SYSTEM FillingCellFixed (* FillingCell (production, OPC UA driven), FillingCellDemo (self-running), SkillBench and PatternDemo run on one FORTE_PC device; PiIoConfig is for a Raspberry Pi *)
  (* Standard: 61499-2 *)
  APPLICATION FillingCell (* Production cell driven over OPC UA (/Objects/FillingCell/Filler). IoBackend 0 = simulated (force Observer.Sim_* ), 1 = GPIO (add PiIoConfig), 2 = Modbus (4diac/tools/cell_sim.py) *)
    FBS
      Boot : iec61499::events::E_RESTART;
      Observer : fillingcell::UNIT_Observer(UaRoot := "/Objects/FillingCell/Filler", UaEnable := TRUE, IoBackend := 0, NeedleUp_Gpio := 'FC_NeedleUp', NeedleUp_Modbus := "modbus[127.0.0.1:1502:1:50:d0:]", NeedleDown_Gpio := 'FC_NeedleDown', NeedleDown_Modbus := "modbus[127.0.0.1:1502:1:50:d1:]", VialPresent_Gpio := 'FC_VialPresent', VialPresent_Modbus := "modbus[127.0.0.1:1502:1:50:d2:]", Stoppered_Gpio := 'FC_Stoppered', Stoppered_Modbus := "modbus[127.0.0.1:1502:1:50:d3:]", Checked_Gpio := 'FC_Checked', Checked_Modbus := "modbus[127.0.0.1:1502:1:50:d4:]", DoorClosed_Gpio := 'FC_DoorClosed', DoorClosed_Modbus := "modbus[127.0.0.1:1502:1:50:d5:]", FilledMl_Gpio := '', FilledMl_Modbus := "modbus[127.0.0.1:1502:1:50:i0:]", Sim_NeedleUp := TRUE, Sim_VialPresent := TRUE, Sim_DoorClosed := TRUE);
      UaFacade : fillingcell::UNIT_Facade(UaRoot := "/Objects/FillingCell/Filler", UaEnable := TRUE);
      Occupation : fillingcell::FC_Occupation;
      Unit : fillingcell::FC_Unit;
      Facade : fillingcell::FC_ProcedureFacade;
    END_FBS
    SUBAPPLICATION EM_Filler (* Equipment module: one composite per skill, chained for status; instances and chain may be changed online while the unit is quiescent *)
      EVENT_INPUT
        INIT;
        UNIT_CTL WITH ControlCode;
        UNIT_STAT WITH UnitRunning, UnitQuiescent, UnitState, Mode, Owner, RemoteAllowed;
        SAMPLE WITH Cell;
        CALL_MoveDown WITH P1_MoveDown, P2_MoveDown, P3_MoveDown, P4_MoveDown;
        CALL_Dose WITH P1_Dose, P2_Dose, P3_Dose, P4_Dose;
        CALL_MoveUp WITH P1_MoveUp, P2_MoveUp, P3_MoveUp, P4_MoveUp;
        CALL_Stopper WITH P1_Stopper, P2_Stopper, P3_Stopper, P4_Stopper;
        CALL_Inspect WITH P1_Inspect, P2_Inspect, P3_Inspect, P4_Inspect;
      END_EVENT
      EVENT_OUTPUT
        INITO;
        STAT_OUT WITH Busy, HeldAll, RunAll;
        DONE_MoveDown;
        DONE_Dose;
        DONE_MoveUp;
        DONE_Stopper;
        DONE_Inspect;
        FAILED_MoveDown WITH CallError_MoveDown;
        FAILED_Dose WITH CallError_Dose;
        FAILED_MoveUp WITH CallError_MoveUp;
        FAILED_Stopper WITH CallError_Stopper;
        FAILED_Inspect WITH CallError_Inspect;
      END_EVENT
      VAR_INPUT
        ControlCode : USINT;
        UnitRunning : BOOL;
        UnitQuiescent : BOOL;
        UnitState : USINT;
        Mode : USINT;
        Owner : UDINT;
        RemoteAllowed : BOOL;
        Cell : fillingcell::ST_CellState;
        P1_MoveDown : LREAL;
        P2_MoveDown : LREAL;
        P3_MoveDown : LREAL;
        P4_MoveDown : LREAL;
        P1_Dose : LREAL;
        P2_Dose : LREAL;
        P3_Dose : LREAL;
        P4_Dose : LREAL;
        P1_MoveUp : LREAL;
        P2_MoveUp : LREAL;
        P3_MoveUp : LREAL;
        P4_MoveUp : LREAL;
        P1_Stopper : LREAL;
        P2_Stopper : LREAL;
        P3_Stopper : LREAL;
        P4_Stopper : LREAL;
        P1_Inspect : LREAL;
        P2_Inspect : LREAL;
        P3_Inspect : LREAL;
        P4_Inspect : LREAL;
      END_VAR
      VAR_OUTPUT
        Busy : BOOL;
        HeldAll : BOOL;
        RunAll : BOOL;
        CallError_MoveDown : UINT;
        CallError_Dose : UINT;
        CallError_MoveUp : UINT;
        CallError_Stopper : UINT;
        CallError_Inspect : UINT;
        Drive_MoveDown : BOOL;
        Drive_Dose : BOOL;
        Drive_MoveUp : BOOL;
        Drive_Stopper : BOOL;
        Drive_Inspect : BOOL;
      END_VAR
      FBS
        MoveDown : fillingcell::SK_MoveDown(UaRoot := "/Objects/FillingCell/Filler/Skills/MoveDown", UaEnable := TRUE, IoBackend := 0, DoGpio := 'FC_MoveDown', DoModbus := "modbus[127.0.0.1:1502:1:0::c0]");
        Dose : fillingcell::SK_Dose(UaRoot := "/Objects/FillingCell/Filler/Skills/Dose", UaEnable := TRUE, IoBackend := 0, DoGpio := 'FC_Dose', DoModbus := "modbus[127.0.0.1:1502:1:0::c1]");
        MoveUp : fillingcell::SK_MoveUp(UaRoot := "/Objects/FillingCell/Filler/Skills/MoveUp", UaEnable := TRUE, IoBackend := 0, DoGpio := 'FC_MoveUp', DoModbus := "modbus[127.0.0.1:1502:1:0::c2]");
        Stopper : fillingcell::SK_Stopper(UaRoot := "/Objects/FillingCell/Filler/Skills/Stopper", UaEnable := TRUE, IoBackend := 0, DoGpio := 'FC_Stopper', DoModbus := "modbus[127.0.0.1:1502:1:0::c3]");
        Inspect : fillingcell::SK_Inspect(UaRoot := "/Objects/FillingCell/Filler/Skills/Inspect", UaEnable := TRUE, IoBackend := 0, DoGpio := 'FC_Inspect', DoModbus := "modbus[127.0.0.1:1502:1:0::c4]");
      END_FBS
      EVENT_CONNECTIONS
        INIT TO MoveDown.INIT;
        MoveDown.INITO TO Dose.INIT;
        MoveDown.STAT_OUT TO Dose.STAT_IN;
        Dose.INITO TO MoveUp.INIT;
        Dose.STAT_OUT TO MoveUp.STAT_IN;
        MoveUp.INITO TO Stopper.INIT;
        MoveUp.STAT_OUT TO Stopper.STAT_IN;
        Stopper.INITO TO Inspect.INIT;
        Stopper.STAT_OUT TO Inspect.STAT_IN;
        Inspect.INITO TO INITO;
        Inspect.STAT_OUT TO STAT_OUT;
        UNIT_CTL TO MoveDown.UNIT_CTL;
        UNIT_STAT TO MoveDown.UNIT_STAT;
        SAMPLE TO MoveDown.SAMPLE;
        CALL_MoveDown TO MoveDown.CALL;
        MoveDown.DONE TO DONE_MoveDown;
        MoveDown.FAILED TO FAILED_MoveDown;
        UNIT_CTL TO Dose.UNIT_CTL;
        UNIT_STAT TO Dose.UNIT_STAT;
        SAMPLE TO Dose.SAMPLE;
        CALL_Dose TO Dose.CALL;
        Dose.DONE TO DONE_Dose;
        Dose.FAILED TO FAILED_Dose;
        UNIT_CTL TO MoveUp.UNIT_CTL;
        UNIT_STAT TO MoveUp.UNIT_STAT;
        SAMPLE TO MoveUp.SAMPLE;
        CALL_MoveUp TO MoveUp.CALL;
        MoveUp.DONE TO DONE_MoveUp;
        MoveUp.FAILED TO FAILED_MoveUp;
        UNIT_CTL TO Stopper.UNIT_CTL;
        UNIT_STAT TO Stopper.UNIT_STAT;
        SAMPLE TO Stopper.SAMPLE;
        CALL_Stopper TO Stopper.CALL;
        Stopper.DONE TO DONE_Stopper;
        Stopper.FAILED TO FAILED_Stopper;
        UNIT_CTL TO Inspect.UNIT_CTL;
        UNIT_STAT TO Inspect.UNIT_STAT;
        SAMPLE TO Inspect.SAMPLE;
        CALL_Inspect TO Inspect.CALL;
        Inspect.DONE TO DONE_Inspect;
        Inspect.FAILED TO FAILED_Inspect;
      END_CONNECTIONS
      DATA_CONNECTIONS
        MoveDown.BusyOut TO Dose.BusyIn;
        MoveDown.HeldOut TO Dose.HeldIn;
        MoveDown.RunOut TO Dose.RunIn;
        Dose.BusyOut TO MoveUp.BusyIn;
        Dose.HeldOut TO MoveUp.HeldIn;
        Dose.RunOut TO MoveUp.RunIn;
        MoveUp.BusyOut TO Stopper.BusyIn;
        MoveUp.HeldOut TO Stopper.HeldIn;
        MoveUp.RunOut TO Stopper.RunIn;
        Stopper.BusyOut TO Inspect.BusyIn;
        Stopper.HeldOut TO Inspect.HeldIn;
        Stopper.RunOut TO Inspect.RunIn;
        Inspect.BusyOut TO Busy;
        Inspect.HeldOut TO HeldAll;
        Inspect.RunOut TO RunAll;
        ControlCode TO MoveDown.ControlCode;
        Cell TO MoveDown.Cell;
        MoveDown.CallError TO CallError_MoveDown;
        MoveDown.Drive TO Drive_MoveDown;
        UnitRunning TO MoveDown.UnitRunning;
        UnitQuiescent TO MoveDown.UnitQuiescent;
        UnitState TO MoveDown.UnitState;
        Mode TO MoveDown.Mode;
        Owner TO MoveDown.Owner;
        RemoteAllowed TO MoveDown.RemoteAllowed;
        P1_MoveDown TO MoveDown.P1;
        P2_MoveDown TO MoveDown.P2;
        P3_MoveDown TO MoveDown.P3;
        P4_MoveDown TO MoveDown.P4;
        ControlCode TO Dose.ControlCode;
        Cell TO Dose.Cell;
        Dose.CallError TO CallError_Dose;
        Dose.Drive TO Drive_Dose;
        UnitRunning TO Dose.UnitRunning;
        UnitQuiescent TO Dose.UnitQuiescent;
        UnitState TO Dose.UnitState;
        Mode TO Dose.Mode;
        Owner TO Dose.Owner;
        RemoteAllowed TO Dose.RemoteAllowed;
        P1_Dose TO Dose.P1;
        P2_Dose TO Dose.P2;
        P3_Dose TO Dose.P3;
        P4_Dose TO Dose.P4;
        ControlCode TO MoveUp.ControlCode;
        Cell TO MoveUp.Cell;
        MoveUp.CallError TO CallError_MoveUp;
        MoveUp.Drive TO Drive_MoveUp;
        UnitRunning TO MoveUp.UnitRunning;
        UnitQuiescent TO MoveUp.UnitQuiescent;
        UnitState TO MoveUp.UnitState;
        Mode TO MoveUp.Mode;
        Owner TO MoveUp.Owner;
        RemoteAllowed TO MoveUp.RemoteAllowed;
        P1_MoveUp TO MoveUp.P1;
        P2_MoveUp TO MoveUp.P2;
        P3_MoveUp TO MoveUp.P3;
        P4_MoveUp TO MoveUp.P4;
        ControlCode TO Stopper.ControlCode;
        Cell TO Stopper.Cell;
        Stopper.CallError TO CallError_Stopper;
        Stopper.Drive TO Drive_Stopper;
        UnitRunning TO Stopper.UnitRunning;
        UnitQuiescent TO Stopper.UnitQuiescent;
        UnitState TO Stopper.UnitState;
        Mode TO Stopper.Mode;
        Owner TO Stopper.Owner;
        RemoteAllowed TO Stopper.RemoteAllowed;
        P1_Stopper TO Stopper.P1;
        P2_Stopper TO Stopper.P2;
        P3_Stopper TO Stopper.P3;
        P4_Stopper TO Stopper.P4;
        ControlCode TO Inspect.ControlCode;
        Cell TO Inspect.Cell;
        Inspect.CallError TO CallError_Inspect;
        Inspect.Drive TO Drive_Inspect;
        UnitRunning TO Inspect.UnitRunning;
        UnitQuiescent TO Inspect.UnitQuiescent;
        UnitState TO Inspect.UnitState;
        Mode TO Inspect.Mode;
        Owner TO Inspect.Owner;
        RemoteAllowed TO Inspect.RemoteAllowed;
        P1_Inspect TO Inspect.P1;
        P2_Inspect TO Inspect.P2;
        P3_Inspect TO Inspect.P3;
        P4_Inspect TO Inspect.P4;
      END_CONNECTIONS
    END_SUBAPPLICATION
    SUBAPPLICATION PROC (* INTENTIONALLY EMPTY: generated procedure (P_* pattern instances) calls skills via CALL_*/DONE_*/FAILED_* *)
      EVENT_INPUT
        START;
        RESET;
        CMD WITH Command;
        DONE_MoveDown;
        DONE_Dose;
        DONE_MoveUp;
        DONE_Stopper;
        DONE_Inspect;
        FAILED_MoveDown WITH CallError_MoveDown;
        FAILED_Dose WITH CallError_Dose;
        FAILED_MoveUp WITH CallError_MoveUp;
        FAILED_Stopper WITH CallError_Stopper;
        FAILED_Inspect WITH CallError_Inspect;
      END_EVENT
      EVENT_OUTPUT
        FINISHED;
        FAILED;
        CALL_MoveDown WITH P1_MoveDown, P2_MoveDown, P3_MoveDown, P4_MoveDown;
        CALL_Dose WITH P1_Dose, P2_Dose, P3_Dose, P4_Dose;
        CALL_MoveUp WITH P1_MoveUp, P2_MoveUp, P3_MoveUp, P4_MoveUp;
        CALL_Stopper WITH P1_Stopper, P2_Stopper, P3_Stopper, P4_Stopper;
        CALL_Inspect WITH P1_Inspect, P2_Inspect, P3_Inspect, P4_Inspect;
      END_EVENT
      VAR_INPUT
        Command : USINT;
        CallError_MoveDown : UINT;
        CallError_Dose : UINT;
        CallError_MoveUp : UINT;
        CallError_Stopper : UINT;
        CallError_Inspect : UINT;
      END_VAR
      VAR_OUTPUT
        P1_MoveDown : LREAL;
        P2_MoveDown : LREAL;
        P3_MoveDown : LREAL;
        P4_MoveDown : LREAL;
        P1_Dose : LREAL;
        P2_Dose : LREAL;
        P3_Dose : LREAL;
        P4_Dose : LREAL;
        P1_MoveUp : LREAL;
        P2_MoveUp : LREAL;
        P3_MoveUp : LREAL;
        P4_MoveUp : LREAL;
        P1_Stopper : LREAL;
        P2_Stopper : LREAL;
        P3_Stopper : LREAL;
        P4_Stopper : LREAL;
        P1_Inspect : LREAL;
        P2_Inspect : LREAL;
        P3_Inspect : LREAL;
        P4_Inspect : LREAL;
      END_VAR
    END_SUBAPPLICATION
    EVENT_CONNECTIONS
      Boot.COLD TO Observer.INIT;
      Boot.WARM TO Observer.INIT;
      Unit.CNF TO EM_Filler.UNIT_STAT;
      Occupation.CNF TO EM_Filler.UNIT_STAT;
      Unit.CONTROL TO EM_Filler.UNIT_CTL;
      EM_Filler.STAT_OUT TO Unit.STATUS;
      Observer.SAMPLE TO EM_Filler.SAMPLE;
      Observer.UNSAFE TO Unit.UNSAFE;
      Unit.PROC_CMD TO Facade.CMD;
      Facade.EXEC TO PROC.CMD;
      Facade.START TO PROC.START;
      Facade.RESET TO PROC.RESET;
      PROC.FINISHED TO Facade.FINISHED;
      PROC.FAILED TO Facade.FAILED;
      Facade.DONE TO Unit.PROC_DONE;
      Facade.FAULT TO Unit.FAULT;
      PROC.CALL_MoveDown TO EM_Filler.CALL_MoveDown;
      EM_Filler.DONE_MoveDown TO PROC.DONE_MoveDown;
      EM_Filler.FAILED_MoveDown TO PROC.FAILED_MoveDown;
      PROC.CALL_Dose TO EM_Filler.CALL_Dose;
      EM_Filler.DONE_Dose TO PROC.DONE_Dose;
      EM_Filler.FAILED_Dose TO PROC.FAILED_Dose;
      PROC.CALL_MoveUp TO EM_Filler.CALL_MoveUp;
      EM_Filler.DONE_MoveUp TO PROC.DONE_MoveUp;
      EM_Filler.FAILED_MoveUp TO PROC.FAILED_MoveUp;
      PROC.CALL_Stopper TO EM_Filler.CALL_Stopper;
      EM_Filler.DONE_Stopper TO PROC.DONE_Stopper;
      EM_Filler.FAILED_Stopper TO PROC.FAILED_Stopper;
      PROC.CALL_Inspect TO EM_Filler.CALL_Inspect;
      EM_Filler.DONE_Inspect TO PROC.DONE_Inspect;
      EM_Filler.FAILED_Inspect TO PROC.FAILED_Inspect;
      Observer.INITO TO UaFacade.INIT;
      UaFacade.INITO TO EM_Filler.INIT;
      UaFacade.U_CMD TO Unit.CMD;
      UaFacade.O_CMD TO Occupation.CMD;
      Unit.CMD_ACK TO UaFacade.U_ACK;
      Unit.CMD_REJ TO UaFacade.U_REJ;
      Occupation.CNF TO UaFacade.O_ACK;
      Occupation.REJECTED TO UaFacade.O_REJ;
      Unit.CNF TO UaFacade.PUB;
      Occupation.CNF TO UaFacade.PUB;
    END_CONNECTIONS
    DATA_CONNECTIONS
      Occupation.Owner TO Unit.Owner;
      Occupation.RemoteAllowed TO Unit.RemoteAllowed;
      Occupation.Owner TO EM_Filler.Owner;
      Occupation.RemoteAllowed TO EM_Filler.RemoteAllowed;
      Unit.Running TO EM_Filler.UnitRunning;
      Unit.Quiescent TO EM_Filler.UnitQuiescent;
      Unit.State TO EM_Filler.UnitState;
      Unit.Mode TO EM_Filler.Mode;
      Unit.ControlCode TO EM_Filler.ControlCode;
      Unit.Quiescent TO Occupation.Quiescent;
      Unit.Quiescent TO Facade.Quiescent;
      EM_Filler.Busy TO Unit.Busy;
      EM_Filler.HeldAll TO Unit.HeldAll;
      EM_Filler.RunAll TO Unit.RunAll;
      Observer.Cell TO EM_Filler.Cell;
      Observer.Safe TO Unit.Safe;
      Unit.ProcedureCommand TO Facade.Command;
      Facade.CommandOut TO PROC.Command;
      Facade.Ready TO Unit.ProcedureReady;
      PROC.P1_MoveDown TO EM_Filler.P1_MoveDown;
      PROC.P2_MoveDown TO EM_Filler.P2_MoveDown;
      PROC.P3_MoveDown TO EM_Filler.P3_MoveDown;
      PROC.P4_MoveDown TO EM_Filler.P4_MoveDown;
      EM_Filler.CallError_MoveDown TO PROC.CallError_MoveDown;
      PROC.P1_Dose TO EM_Filler.P1_Dose;
      PROC.P2_Dose TO EM_Filler.P2_Dose;
      PROC.P3_Dose TO EM_Filler.P3_Dose;
      PROC.P4_Dose TO EM_Filler.P4_Dose;
      EM_Filler.CallError_Dose TO PROC.CallError_Dose;
      PROC.P1_MoveUp TO EM_Filler.P1_MoveUp;
      PROC.P2_MoveUp TO EM_Filler.P2_MoveUp;
      PROC.P3_MoveUp TO EM_Filler.P3_MoveUp;
      PROC.P4_MoveUp TO EM_Filler.P4_MoveUp;
      EM_Filler.CallError_MoveUp TO PROC.CallError_MoveUp;
      PROC.P1_Stopper TO EM_Filler.P1_Stopper;
      PROC.P2_Stopper TO EM_Filler.P2_Stopper;
      PROC.P3_Stopper TO EM_Filler.P3_Stopper;
      PROC.P4_Stopper TO EM_Filler.P4_Stopper;
      EM_Filler.CallError_Stopper TO PROC.CallError_Stopper;
      PROC.P1_Inspect TO EM_Filler.P1_Inspect;
      PROC.P2_Inspect TO EM_Filler.P2_Inspect;
      PROC.P3_Inspect TO EM_Filler.P3_Inspect;
      PROC.P4_Inspect TO EM_Filler.P4_Inspect;
      EM_Filler.CallError_Inspect TO PROC.CallError_Inspect;
      UaFacade.Requester TO Unit.Requester;
      UaFacade.Requester TO Occupation.Requester;
      UaFacade.U_Code TO Unit.Command;
      UaFacade.U_Mode TO Unit.RequestedMode;
      UaFacade.O_Code TO Occupation.Command;
      Unit.State TO UaFacade.UnitState;
      Unit.Mode TO UaFacade.UnitMode;
      Occupation.State TO UaFacade.OccState;
      Occupation.Owner TO UaFacade.Owner;
    END_CONNECTIONS
  END_APPLICATION
  APPLICATION FillingCellDemo (* Self-running demo: plant model and automatic operator cycle the whole cell through the PROC procedure; watch Operator.Cycles, Unit.State, Plant.* in the IDE monitoring (no OPC UA: FORTE 3.3 serves OPC UA for one resource only, used by FillingCell) *)
    FBS
      Boot : iec61499::events::E_RESTART;
      Observer : fillingcell::UNIT_Observer(UaRoot := "/Objects/Demo/Filler", UaEnable := FALSE, IoBackend := 0, CycleTime := T#50ms);
      Occupation : fillingcell::FC_Occupation;
      Unit : fillingcell::FC_Unit;
      Facade : fillingcell::FC_ProcedureFacade(Installed := TRUE);
      Plant : fillingcell::DEMO_Plant;
      PlantClock : iec61499::events::E_CYCLE(DT := T#20ms);
      Operator : fillingcell::DEMO_Operator;
      OpDelay : iec61499::events::E_DELAY;
    END_FBS
    SUBAPPLICATION EM_Filler (* Equipment module: one composite per skill, chained for status; instances and chain may be changed online while the unit is quiescent *)
      EVENT_INPUT
        INIT;
        UNIT_CTL WITH ControlCode;
        UNIT_STAT WITH UnitRunning, UnitQuiescent, UnitState, Mode, Owner, RemoteAllowed;
        SAMPLE WITH Cell;
        CALL_MoveDown WITH P1_MoveDown, P2_MoveDown, P3_MoveDown, P4_MoveDown;
        CALL_Dose WITH P1_Dose, P2_Dose, P3_Dose, P4_Dose;
        CALL_MoveUp WITH P1_MoveUp, P2_MoveUp, P3_MoveUp, P4_MoveUp;
        CALL_Stopper WITH P1_Stopper, P2_Stopper, P3_Stopper, P4_Stopper;
        CALL_Inspect WITH P1_Inspect, P2_Inspect, P3_Inspect, P4_Inspect;
      END_EVENT
      EVENT_OUTPUT
        INITO;
        STAT_OUT WITH Busy, HeldAll, RunAll;
        DONE_MoveDown;
        DONE_Dose;
        DONE_MoveUp;
        DONE_Stopper;
        DONE_Inspect;
        FAILED_MoveDown WITH CallError_MoveDown;
        FAILED_Dose WITH CallError_Dose;
        FAILED_MoveUp WITH CallError_MoveUp;
        FAILED_Stopper WITH CallError_Stopper;
        FAILED_Inspect WITH CallError_Inspect;
      END_EVENT
      VAR_INPUT
        ControlCode : USINT;
        UnitRunning : BOOL;
        UnitQuiescent : BOOL;
        UnitState : USINT;
        Mode : USINT;
        Owner : UDINT;
        RemoteAllowed : BOOL;
        Cell : fillingcell::ST_CellState;
        P1_MoveDown : LREAL;
        P2_MoveDown : LREAL;
        P3_MoveDown : LREAL;
        P4_MoveDown : LREAL;
        P1_Dose : LREAL;
        P2_Dose : LREAL;
        P3_Dose : LREAL;
        P4_Dose : LREAL;
        P1_MoveUp : LREAL;
        P2_MoveUp : LREAL;
        P3_MoveUp : LREAL;
        P4_MoveUp : LREAL;
        P1_Stopper : LREAL;
        P2_Stopper : LREAL;
        P3_Stopper : LREAL;
        P4_Stopper : LREAL;
        P1_Inspect : LREAL;
        P2_Inspect : LREAL;
        P3_Inspect : LREAL;
        P4_Inspect : LREAL;
      END_VAR
      VAR_OUTPUT
        Busy : BOOL;
        HeldAll : BOOL;
        RunAll : BOOL;
        CallError_MoveDown : UINT;
        CallError_Dose : UINT;
        CallError_MoveUp : UINT;
        CallError_Stopper : UINT;
        CallError_Inspect : UINT;
        Drive_MoveDown : BOOL;
        Drive_Dose : BOOL;
        Drive_MoveUp : BOOL;
        Drive_Stopper : BOOL;
        Drive_Inspect : BOOL;
      END_VAR
      FBS
        MoveDown : fillingcell::SK_MoveDown(UaRoot := "/Objects/Demo/Filler/Skills/MoveDown", UaEnable := FALSE, IoBackend := 0);
        Dose : fillingcell::SK_Dose(UaRoot := "/Objects/Demo/Filler/Skills/Dose", UaEnable := FALSE, IoBackend := 0);
        MoveUp : fillingcell::SK_MoveUp(UaRoot := "/Objects/Demo/Filler/Skills/MoveUp", UaEnable := FALSE, IoBackend := 0);
        Stopper : fillingcell::SK_Stopper(UaRoot := "/Objects/Demo/Filler/Skills/Stopper", UaEnable := FALSE, IoBackend := 0);
        Inspect : fillingcell::SK_Inspect(UaRoot := "/Objects/Demo/Filler/Skills/Inspect", UaEnable := FALSE, IoBackend := 0);
      END_FBS
      EVENT_CONNECTIONS
        INIT TO MoveDown.INIT;
        MoveDown.INITO TO Dose.INIT;
        MoveDown.STAT_OUT TO Dose.STAT_IN;
        Dose.INITO TO MoveUp.INIT;
        Dose.STAT_OUT TO MoveUp.STAT_IN;
        MoveUp.INITO TO Stopper.INIT;
        MoveUp.STAT_OUT TO Stopper.STAT_IN;
        Stopper.INITO TO Inspect.INIT;
        Stopper.STAT_OUT TO Inspect.STAT_IN;
        Inspect.INITO TO INITO;
        Inspect.STAT_OUT TO STAT_OUT;
        UNIT_CTL TO MoveDown.UNIT_CTL;
        UNIT_STAT TO MoveDown.UNIT_STAT;
        SAMPLE TO MoveDown.SAMPLE;
        CALL_MoveDown TO MoveDown.CALL;
        MoveDown.DONE TO DONE_MoveDown;
        MoveDown.FAILED TO FAILED_MoveDown;
        UNIT_CTL TO Dose.UNIT_CTL;
        UNIT_STAT TO Dose.UNIT_STAT;
        SAMPLE TO Dose.SAMPLE;
        CALL_Dose TO Dose.CALL;
        Dose.DONE TO DONE_Dose;
        Dose.FAILED TO FAILED_Dose;
        UNIT_CTL TO MoveUp.UNIT_CTL;
        UNIT_STAT TO MoveUp.UNIT_STAT;
        SAMPLE TO MoveUp.SAMPLE;
        CALL_MoveUp TO MoveUp.CALL;
        MoveUp.DONE TO DONE_MoveUp;
        MoveUp.FAILED TO FAILED_MoveUp;
        UNIT_CTL TO Stopper.UNIT_CTL;
        UNIT_STAT TO Stopper.UNIT_STAT;
        SAMPLE TO Stopper.SAMPLE;
        CALL_Stopper TO Stopper.CALL;
        Stopper.DONE TO DONE_Stopper;
        Stopper.FAILED TO FAILED_Stopper;
        UNIT_CTL TO Inspect.UNIT_CTL;
        UNIT_STAT TO Inspect.UNIT_STAT;
        SAMPLE TO Inspect.SAMPLE;
        CALL_Inspect TO Inspect.CALL;
        Inspect.DONE TO DONE_Inspect;
        Inspect.FAILED TO FAILED_Inspect;
      END_CONNECTIONS
      DATA_CONNECTIONS
        MoveDown.BusyOut TO Dose.BusyIn;
        MoveDown.HeldOut TO Dose.HeldIn;
        MoveDown.RunOut TO Dose.RunIn;
        Dose.BusyOut TO MoveUp.BusyIn;
        Dose.HeldOut TO MoveUp.HeldIn;
        Dose.RunOut TO MoveUp.RunIn;
        MoveUp.BusyOut TO Stopper.BusyIn;
        MoveUp.HeldOut TO Stopper.HeldIn;
        MoveUp.RunOut TO Stopper.RunIn;
        Stopper.BusyOut TO Inspect.BusyIn;
        Stopper.HeldOut TO Inspect.HeldIn;
        Stopper.RunOut TO Inspect.RunIn;
        Inspect.BusyOut TO Busy;
        Inspect.HeldOut TO HeldAll;
        Inspect.RunOut TO RunAll;
        ControlCode TO MoveDown.ControlCode;
        Cell TO MoveDown.Cell;
        MoveDown.CallError TO CallError_MoveDown;
        MoveDown.Drive TO Drive_MoveDown;
        UnitRunning TO MoveDown.UnitRunning;
        UnitQuiescent TO MoveDown.UnitQuiescent;
        UnitState TO MoveDown.UnitState;
        Mode TO MoveDown.Mode;
        Owner TO MoveDown.Owner;
        RemoteAllowed TO MoveDown.RemoteAllowed;
        P1_MoveDown TO MoveDown.P1;
        P2_MoveDown TO MoveDown.P2;
        P3_MoveDown TO MoveDown.P3;
        P4_MoveDown TO MoveDown.P4;
        ControlCode TO Dose.ControlCode;
        Cell TO Dose.Cell;
        Dose.CallError TO CallError_Dose;
        Dose.Drive TO Drive_Dose;
        UnitRunning TO Dose.UnitRunning;
        UnitQuiescent TO Dose.UnitQuiescent;
        UnitState TO Dose.UnitState;
        Mode TO Dose.Mode;
        Owner TO Dose.Owner;
        RemoteAllowed TO Dose.RemoteAllowed;
        P1_Dose TO Dose.P1;
        P2_Dose TO Dose.P2;
        P3_Dose TO Dose.P3;
        P4_Dose TO Dose.P4;
        ControlCode TO MoveUp.ControlCode;
        Cell TO MoveUp.Cell;
        MoveUp.CallError TO CallError_MoveUp;
        MoveUp.Drive TO Drive_MoveUp;
        UnitRunning TO MoveUp.UnitRunning;
        UnitQuiescent TO MoveUp.UnitQuiescent;
        UnitState TO MoveUp.UnitState;
        Mode TO MoveUp.Mode;
        Owner TO MoveUp.Owner;
        RemoteAllowed TO MoveUp.RemoteAllowed;
        P1_MoveUp TO MoveUp.P1;
        P2_MoveUp TO MoveUp.P2;
        P3_MoveUp TO MoveUp.P3;
        P4_MoveUp TO MoveUp.P4;
        ControlCode TO Stopper.ControlCode;
        Cell TO Stopper.Cell;
        Stopper.CallError TO CallError_Stopper;
        Stopper.Drive TO Drive_Stopper;
        UnitRunning TO Stopper.UnitRunning;
        UnitQuiescent TO Stopper.UnitQuiescent;
        UnitState TO Stopper.UnitState;
        Mode TO Stopper.Mode;
        Owner TO Stopper.Owner;
        RemoteAllowed TO Stopper.RemoteAllowed;
        P1_Stopper TO Stopper.P1;
        P2_Stopper TO Stopper.P2;
        P3_Stopper TO Stopper.P3;
        P4_Stopper TO Stopper.P4;
        ControlCode TO Inspect.ControlCode;
        Cell TO Inspect.Cell;
        Inspect.CallError TO CallError_Inspect;
        Inspect.Drive TO Drive_Inspect;
        UnitRunning TO Inspect.UnitRunning;
        UnitQuiescent TO Inspect.UnitQuiescent;
        UnitState TO Inspect.UnitState;
        Mode TO Inspect.Mode;
        Owner TO Inspect.Owner;
        RemoteAllowed TO Inspect.RemoteAllowed;
        P1_Inspect TO Inspect.P1;
        P2_Inspect TO Inspect.P2;
        P3_Inspect TO Inspect.P3;
        P4_Inspect TO Inspect.P4;
      END_CONNECTIONS
    END_SUBAPPLICATION
    SUBAPPLICATION PROC (* Demo procedure: MoveDown, Dose x2 (P_Loop), MoveUp, Stopper, Inspect *)
      EVENT_INPUT
        START;
        RESET;
        CMD WITH Command;
        DONE_MoveDown;
        DONE_Dose;
        DONE_MoveUp;
        DONE_Stopper;
        DONE_Inspect;
        FAILED_MoveDown WITH CallError_MoveDown;
        FAILED_Dose WITH CallError_Dose;
        FAILED_MoveUp WITH CallError_MoveUp;
        FAILED_Stopper WITH CallError_Stopper;
        FAILED_Inspect WITH CallError_Inspect;
      END_EVENT
      EVENT_OUTPUT
        FINISHED;
        FAILED;
        CALL_MoveDown WITH P1_MoveDown, P2_MoveDown, P3_MoveDown, P4_MoveDown;
        CALL_Dose WITH P1_Dose, P2_Dose, P3_Dose, P4_Dose;
        CALL_MoveUp WITH P1_MoveUp, P2_MoveUp, P3_MoveUp, P4_MoveUp;
        CALL_Stopper WITH P1_Stopper, P2_Stopper, P3_Stopper, P4_Stopper;
        CALL_Inspect WITH P1_Inspect, P2_Inspect, P3_Inspect, P4_Inspect;
      END_EVENT
      VAR_INPUT
        Command : USINT;
        CallError_MoveDown : UINT;
        CallError_Dose : UINT;
        CallError_MoveUp : UINT;
        CallError_Stopper : UINT;
        CallError_Inspect : UINT;
      END_VAR
      VAR_OUTPUT
        P1_MoveDown : LREAL;
        P2_MoveDown : LREAL;
        P3_MoveDown : LREAL;
        P4_MoveDown : LREAL;
        P1_Dose : LREAL;
        P2_Dose : LREAL;
        P3_Dose : LREAL;
        P4_Dose : LREAL;
        P1_MoveUp : LREAL;
        P2_MoveUp : LREAL;
        P3_MoveUp : LREAL;
        P4_MoveUp : LREAL;
        P1_Stopper : LREAL;
        P2_Stopper : LREAL;
        P3_Stopper : LREAL;
        P4_Stopper : LREAL;
        P1_Inspect : LREAL;
        P2_Inspect : LREAL;
        P3_Inspect : LREAL;
        P4_Inspect : LREAL;
      END_VAR
      FBS
        MoveDown : fillingcell::P_Call;
        Dose : fillingcell::P_Call(P1 := 0.3);
        MoveUp : fillingcell::P_Call;
        Stopper : fillingcell::P_Call;
        Inspect : fillingcell::P_Call;
        DoseLoop : fillingcell::P_Loop(Count := 2);
      END_FBS
      EVENT_CONNECTIONS
        START TO MoveDown.EI;
        MoveDown.EO TO DoseLoop.EI;
        DoseLoop.BODY TO Dose.EI;
        Dose.EO TO DoseLoop.NEXT;
        DoseLoop.EO TO MoveUp.EI;
        MoveUp.EO TO Stopper.EI;
        Stopper.EO TO Inspect.EI;
        Inspect.EO TO FINISHED;
        RESET TO DoseLoop.RESET;
        MoveDown.CALL TO CALL_MoveDown;
        DONE_MoveDown TO MoveDown.DONE;
        FAILED_MoveDown TO MoveDown.FAILED;
        MoveDown.ERR TO FAILED;
        RESET TO MoveDown.RESET;
        Dose.CALL TO CALL_Dose;
        DONE_Dose TO Dose.DONE;
        FAILED_Dose TO Dose.FAILED;
        Dose.ERR TO FAILED;
        RESET TO Dose.RESET;
        MoveUp.CALL TO CALL_MoveUp;
        DONE_MoveUp TO MoveUp.DONE;
        FAILED_MoveUp TO MoveUp.FAILED;
        MoveUp.ERR TO FAILED;
        RESET TO MoveUp.RESET;
        Stopper.CALL TO CALL_Stopper;
        DONE_Stopper TO Stopper.DONE;
        FAILED_Stopper TO Stopper.FAILED;
        Stopper.ERR TO FAILED;
        RESET TO Stopper.RESET;
        Inspect.CALL TO CALL_Inspect;
        DONE_Inspect TO Inspect.DONE;
        FAILED_Inspect TO Inspect.FAILED;
        Inspect.ERR TO FAILED;
        RESET TO Inspect.RESET;
      END_CONNECTIONS
      DATA_CONNECTIONS
        Dose.CP1 TO P1_Dose;
        CallError_MoveDown TO MoveDown.CallError;
        CallError_Dose TO Dose.CallError;
        CallError_MoveUp TO MoveUp.CallError;
        CallError_Stopper TO Stopper.CallError;
        CallError_Inspect TO Inspect.CallError;
      END_CONNECTIONS
    END_SUBAPPLICATION
    EVENT_CONNECTIONS
      Boot.COLD TO Observer.INIT;
      Boot.WARM TO Observer.INIT;
      Unit.CNF TO EM_Filler.UNIT_STAT;
      Occupation.CNF TO EM_Filler.UNIT_STAT;
      Unit.CONTROL TO EM_Filler.UNIT_CTL;
      EM_Filler.STAT_OUT TO Unit.STATUS;
      Observer.SAMPLE TO EM_Filler.SAMPLE;
      Observer.UNSAFE TO Unit.UNSAFE;
      Unit.PROC_CMD TO Facade.CMD;
      Facade.EXEC TO PROC.CMD;
      Facade.START TO PROC.START;
      Facade.RESET TO PROC.RESET;
      PROC.FINISHED TO Facade.FINISHED;
      PROC.FAILED TO Facade.FAILED;
      Facade.DONE TO Unit.PROC_DONE;
      Facade.FAULT TO Unit.FAULT;
      PROC.CALL_MoveDown TO EM_Filler.CALL_MoveDown;
      EM_Filler.DONE_MoveDown TO PROC.DONE_MoveDown;
      EM_Filler.FAILED_MoveDown TO PROC.FAILED_MoveDown;
      PROC.CALL_Dose TO EM_Filler.CALL_Dose;
      EM_Filler.DONE_Dose TO PROC.DONE_Dose;
      EM_Filler.FAILED_Dose TO PROC.FAILED_Dose;
      PROC.CALL_MoveUp TO EM_Filler.CALL_MoveUp;
      EM_Filler.DONE_MoveUp TO PROC.DONE_MoveUp;
      EM_Filler.FAILED_MoveUp TO PROC.FAILED_MoveUp;
      PROC.CALL_Stopper TO EM_Filler.CALL_Stopper;
      EM_Filler.DONE_Stopper TO PROC.DONE_Stopper;
      EM_Filler.FAILED_Stopper TO PROC.FAILED_Stopper;
      PROC.CALL_Inspect TO EM_Filler.CALL_Inspect;
      EM_Filler.DONE_Inspect TO PROC.DONE_Inspect;
      EM_Filler.FAILED_Inspect TO PROC.FAILED_Inspect;
      Boot.COLD TO Plant.INIT;
      Boot.WARM TO Plant.INIT;
      Boot.COLD TO PlantClock.START;
      Boot.WARM TO PlantClock.START;
      PlantClock.EO TO Plant.TICK;
      Plant.CNF TO Observer.SIM;
      Observer.INITO TO EM_Filler.INIT;
      EM_Filler.INITO TO Facade.CONFIG;
      Facade.CNF TO Operator.START;
      Operator.O_CMD TO Occupation.CMD;
      Operator.U_CMD TO Unit.CMD;
      Operator.NEW_VIAL TO Plant.NEW_VIAL;
      Operator.WAIT TO OpDelay.START;
      OpDelay.EO TO Operator.TIMER;
      Unit.CNF TO Operator.UNIT;
      Unit.CMD_REJ TO Operator.REJ;
    END_CONNECTIONS
    DATA_CONNECTIONS
      Occupation.Owner TO Unit.Owner;
      Occupation.RemoteAllowed TO Unit.RemoteAllowed;
      Occupation.Owner TO EM_Filler.Owner;
      Occupation.RemoteAllowed TO EM_Filler.RemoteAllowed;
      Unit.Running TO EM_Filler.UnitRunning;
      Unit.Quiescent TO EM_Filler.UnitQuiescent;
      Unit.State TO EM_Filler.UnitState;
      Unit.Mode TO EM_Filler.Mode;
      Unit.ControlCode TO EM_Filler.ControlCode;
      Unit.Quiescent TO Occupation.Quiescent;
      Unit.Quiescent TO Facade.Quiescent;
      EM_Filler.Busy TO Unit.Busy;
      EM_Filler.HeldAll TO Unit.HeldAll;
      EM_Filler.RunAll TO Unit.RunAll;
      Observer.Cell TO EM_Filler.Cell;
      Observer.Safe TO Unit.Safe;
      Unit.ProcedureCommand TO Facade.Command;
      Facade.CommandOut TO PROC.Command;
      Facade.Ready TO Unit.ProcedureReady;
      PROC.P1_MoveDown TO EM_Filler.P1_MoveDown;
      PROC.P2_MoveDown TO EM_Filler.P2_MoveDown;
      PROC.P3_MoveDown TO EM_Filler.P3_MoveDown;
      PROC.P4_MoveDown TO EM_Filler.P4_MoveDown;
      EM_Filler.CallError_MoveDown TO PROC.CallError_MoveDown;
      PROC.P1_Dose TO EM_Filler.P1_Dose;
      PROC.P2_Dose TO EM_Filler.P2_Dose;
      PROC.P3_Dose TO EM_Filler.P3_Dose;
      PROC.P4_Dose TO EM_Filler.P4_Dose;
      EM_Filler.CallError_Dose TO PROC.CallError_Dose;
      PROC.P1_MoveUp TO EM_Filler.P1_MoveUp;
      PROC.P2_MoveUp TO EM_Filler.P2_MoveUp;
      PROC.P3_MoveUp TO EM_Filler.P3_MoveUp;
      PROC.P4_MoveUp TO EM_Filler.P4_MoveUp;
      EM_Filler.CallError_MoveUp TO PROC.CallError_MoveUp;
      PROC.P1_Stopper TO EM_Filler.P1_Stopper;
      PROC.P2_Stopper TO EM_Filler.P2_Stopper;
      PROC.P3_Stopper TO EM_Filler.P3_Stopper;
      PROC.P4_Stopper TO EM_Filler.P4_Stopper;
      EM_Filler.CallError_Stopper TO PROC.CallError_Stopper;
      PROC.P1_Inspect TO EM_Filler.P1_Inspect;
      PROC.P2_Inspect TO EM_Filler.P2_Inspect;
      PROC.P3_Inspect TO EM_Filler.P3_Inspect;
      PROC.P4_Inspect TO EM_Filler.P4_Inspect;
      EM_Filler.CallError_Inspect TO PROC.CallError_Inspect;
      Operator.Requester TO Unit.Requester;
      Operator.Requester TO Occupation.Requester;
      Operator.U_Code TO Unit.Command;
      Operator.U_Mode TO Unit.RequestedMode;
      Operator.O_Code TO Occupation.Command;
      Unit.State TO Operator.UnitState;
      Operator.Delay TO OpDelay.DT;
      Plant.NeedleUp TO Observer.Sim_NeedleUp;
      Plant.NeedleDown TO Observer.Sim_NeedleDown;
      Plant.VialPresent TO Observer.Sim_VialPresent;
      Plant.FilledMl TO Observer.Sim_FilledMl;
      Plant.Stoppered TO Observer.Sim_Stoppered;
      Plant.Checked TO Observer.Sim_Checked;
      Plant.DoorClosed TO Observer.Sim_DoorClosed;
      EM_Filler.Drive_MoveDown TO Plant.DriveMoveDown;
      EM_Filler.Drive_Dose TO Plant.DriveDose;
      EM_Filler.Drive_MoveUp TO Plant.DriveMoveUp;
      EM_Filler.Drive_Stopper TO Plant.DriveStopper;
      EM_Filler.Drive_Inspect TO Plant.DriveInspect;
    END_CONNECTIONS
  END_APPLICATION
  APPLICATION SkillBench (* Demo: SK_Dose is called periodically with P1 = 0.3 mL; watch Dose.State, Plant.FilledMl, Done.CV and Failed.CV in the IDE monitoring *)
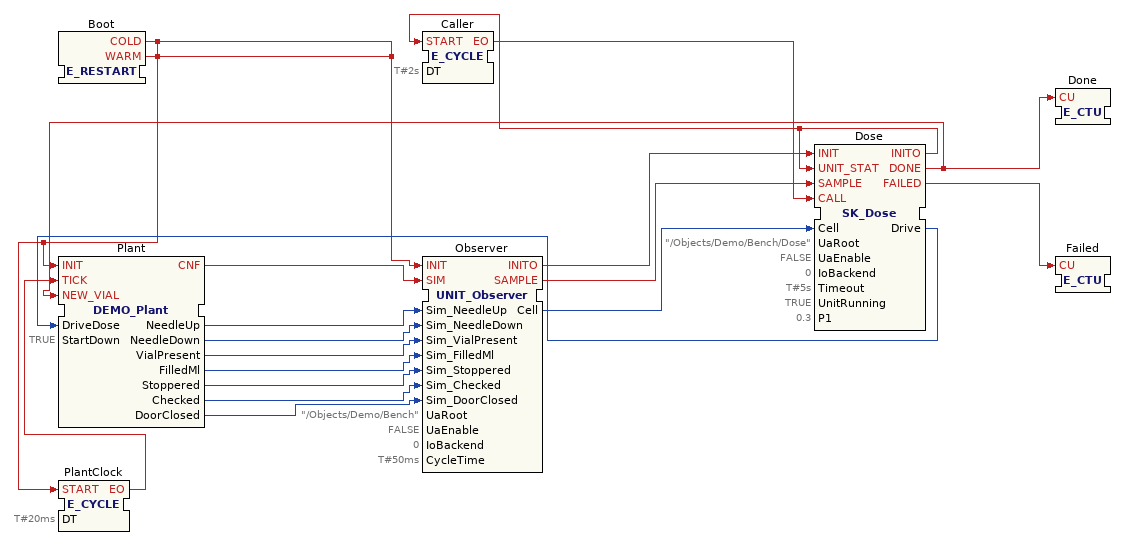
    FBS
      Boot : iec61499::events::E_RESTART;
      Plant : fillingcell::DEMO_Plant(StartDown := TRUE);
      PlantClock : iec61499::events::E_CYCLE(DT := T#20ms);
      Observer : fillingcell::UNIT_Observer(UaRoot := "/Objects/Demo/Bench", UaEnable := FALSE, IoBackend := 0, CycleTime := T#50ms);
      Dose : fillingcell::SK_Dose(UaRoot := "/Objects/Demo/Bench/Dose", UaEnable := FALSE, IoBackend := 0, Timeout := T#5s, UnitRunning := TRUE, P1 := 0.3);
      Caller : iec61499::events::E_CYCLE(DT := T#2s);
      Done : iec61499::events::E_CTU;
      Failed : iec61499::events::E_CTU;
    END_FBS
    EVENT_CONNECTIONS
      Boot.COLD TO Plant.INIT;
      Boot.WARM TO Plant.INIT;
      Boot.COLD TO PlantClock.START;
      Boot.WARM TO PlantClock.START;
      Boot.COLD TO Observer.INIT;
      Boot.WARM TO Observer.INIT;
      PlantClock.EO TO Plant.TICK;
      Plant.CNF TO Observer.SIM;
      Observer.INITO TO Dose.INIT;
      Dose.INITO TO Dose.UNIT_STAT;
      Dose.INITO TO Caller.START;
      Observer.SAMPLE TO Dose.SAMPLE;
      Caller.EO TO Dose.CALL;
      Dose.DONE TO Done.CU;
      Dose.DONE TO Plant.NEW_VIAL;
      Dose.FAILED TO Failed.CU;
    END_CONNECTIONS
    DATA_CONNECTIONS
      Plant.NeedleUp TO Observer.Sim_NeedleUp;
      Plant.NeedleDown TO Observer.Sim_NeedleDown;
      Plant.VialPresent TO Observer.Sim_VialPresent;
      Plant.FilledMl TO Observer.Sim_FilledMl;
      Plant.Stoppered TO Observer.Sim_Stoppered;
      Plant.Checked TO Observer.Sim_Checked;
      Plant.DoorClosed TO Observer.Sim_DoorClosed;
      Observer.Cell TO Dose.Cell;
      Dose.Drive TO Plant.DriveDose;
    END_CONNECTIONS
  END_APPLICATION
  APPLICATION PatternDemo (* Demo of the procedure patterns: every 3 s a fork waits 0.3 s and 0.8 s, the join starts a 3-iteration loop, then a choice alternates; watch the Ctu* counters *)
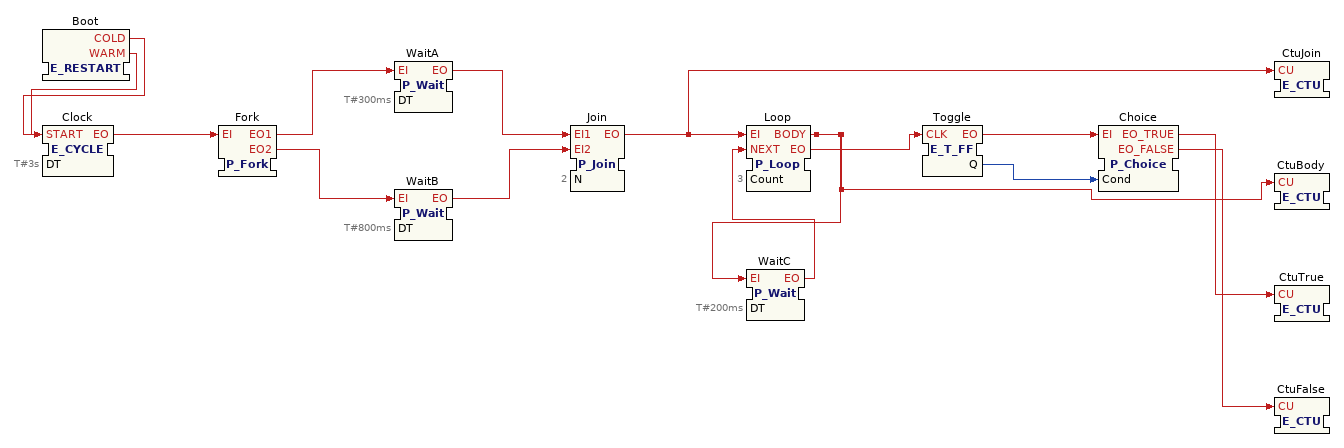
    FBS
      Boot : iec61499::events::E_RESTART;
      Clock : iec61499::events::E_CYCLE(DT := T#3s);
      Fork : fillingcell::P_Fork;
      WaitA : fillingcell::P_Wait(DT := T#300ms);
      WaitB : fillingcell::P_Wait(DT := T#800ms);
      Join : fillingcell::P_Join(N := 2);
      Loop : fillingcell::P_Loop(Count := 3);
      WaitC : fillingcell::P_Wait(DT := T#200ms);
      Toggle : iec61499::events::E_T_FF;
      Choice : fillingcell::P_Choice;
      CtuJoin : iec61499::events::E_CTU;
      CtuBody : iec61499::events::E_CTU;
      CtuTrue : iec61499::events::E_CTU;
      CtuFalse : iec61499::events::E_CTU;
    END_FBS
    EVENT_CONNECTIONS
      Boot.COLD TO Clock.START;
      Boot.WARM TO Clock.START;
      Clock.EO TO Fork.EI;
      Fork.EO1 TO WaitA.EI;
      Fork.EO2 TO WaitB.EI;
      WaitA.EO TO Join.EI1;
      WaitB.EO TO Join.EI2;
      Join.EO TO CtuJoin.CU;
      Join.EO TO Loop.EI;
      Loop.BODY TO WaitC.EI;
      Loop.BODY TO CtuBody.CU;
      WaitC.EO TO Loop.NEXT;
      Loop.EO TO Toggle.CLK;
      Toggle.EO TO Choice.EI;
      Choice.EO_TRUE TO CtuTrue.CU;
      Choice.EO_FALSE TO CtuFalse.CU;
    END_CONNECTIONS
    DATA_CONNECTIONS
      Toggle.Q TO Choice.Cond;
    END_CONNECTIONS
  END_APPLICATION
  APPLICATION PiIoConfig (* GPIOChip line configuration for a Raspberry Pi; handle names match IX/QX PARAMS in FillingCell. Map it together with FillingCell (IoBackend = 1) onto a Pi device *)
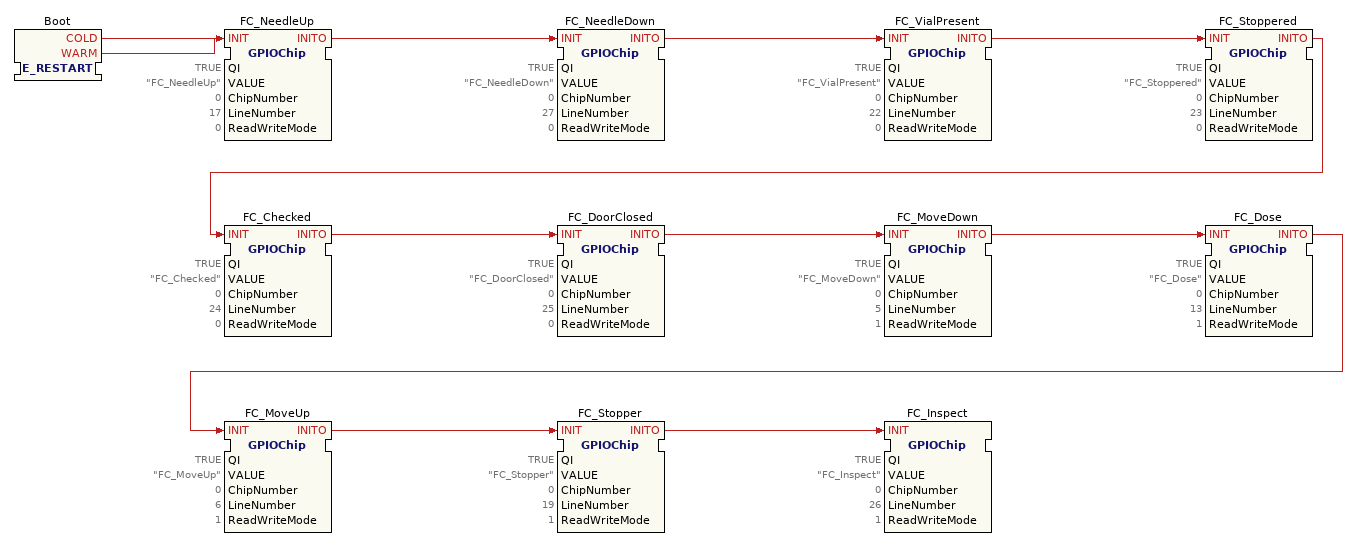
    FBS
      Boot : iec61499::events::E_RESTART;
      FC_NeedleUp : eclipse4diac::io::gpiochip::GPIOChip(QI := TRUE, VALUE := "FC_NeedleUp", ChipNumber := 0, LineNumber := 17, ReadWriteMode := 0);
      FC_NeedleDown : eclipse4diac::io::gpiochip::GPIOChip(QI := TRUE, VALUE := "FC_NeedleDown", ChipNumber := 0, LineNumber := 27, ReadWriteMode := 0);
      FC_VialPresent : eclipse4diac::io::gpiochip::GPIOChip(QI := TRUE, VALUE := "FC_VialPresent", ChipNumber := 0, LineNumber := 22, ReadWriteMode := 0);
      FC_Stoppered : eclipse4diac::io::gpiochip::GPIOChip(QI := TRUE, VALUE := "FC_Stoppered", ChipNumber := 0, LineNumber := 23, ReadWriteMode := 0);
      FC_Checked : eclipse4diac::io::gpiochip::GPIOChip(QI := TRUE, VALUE := "FC_Checked", ChipNumber := 0, LineNumber := 24, ReadWriteMode := 0);
      FC_DoorClosed : eclipse4diac::io::gpiochip::GPIOChip(QI := TRUE, VALUE := "FC_DoorClosed", ChipNumber := 0, LineNumber := 25, ReadWriteMode := 0);
      FC_MoveDown : eclipse4diac::io::gpiochip::GPIOChip(QI := TRUE, VALUE := "FC_MoveDown", ChipNumber := 0, LineNumber := 5, ReadWriteMode := 1);
      FC_Dose : eclipse4diac::io::gpiochip::GPIOChip(QI := TRUE, VALUE := "FC_Dose", ChipNumber := 0, LineNumber := 13, ReadWriteMode := 1);
      FC_MoveUp : eclipse4diac::io::gpiochip::GPIOChip(QI := TRUE, VALUE := "FC_MoveUp", ChipNumber := 0, LineNumber := 6, ReadWriteMode := 1);
      FC_Stopper : eclipse4diac::io::gpiochip::GPIOChip(QI := TRUE, VALUE := "FC_Stopper", ChipNumber := 0, LineNumber := 19, ReadWriteMode := 1);
      FC_Inspect : eclipse4diac::io::gpiochip::GPIOChip(QI := TRUE, VALUE := "FC_Inspect", ChipNumber := 0, LineNumber := 26, ReadWriteMode := 1);
    END_FBS
    EVENT_CONNECTIONS
      Boot.COLD TO FC_NeedleUp.INIT;
      Boot.WARM TO FC_NeedleUp.INIT;
      FC_NeedleUp.INITO TO FC_NeedleDown.INIT;
      FC_NeedleDown.INITO TO FC_VialPresent.INIT;
      FC_VialPresent.INITO TO FC_Stoppered.INIT;
      FC_Stoppered.INITO TO FC_Checked.INIT;
      FC_Checked.INITO TO FC_DoorClosed.INIT;
      FC_DoorClosed.INITO TO FC_MoveDown.INIT;
      FC_MoveDown.INITO TO FC_Dose.INIT;
      FC_Dose.INITO TO FC_MoveUp.INIT;
      FC_MoveUp.INITO TO FC_Stopper.INIT;
      FC_Stopper.INITO TO FC_Inspect.INIT;
    END_CONNECTIONS
  END_APPLICATION
  DEVICE FORTE_PC : iec61499::system::FORTE_PC(MGR_ID := "localhost:61499")
    {SET_ATTRIBUTE(Profile, HOLOBLOC)} (* device profile *)
    RESOURCE RES : iec61499::system::EMB_RES
      FBS
        Boot : iec61499::events::E_RESTART;
        Observer : fillingcell::UNIT_Observer(UaRoot := "/Objects/FillingCell/Filler", UaEnable := TRUE, IoBackend := 0, NeedleUp_Gpio := 'FC_NeedleUp', NeedleUp_Modbus := "modbus[127.0.0.1:1502:1:50:d0:]", NeedleDown_Gpio := 'FC_NeedleDown', NeedleDown_Modbus := "modbus[127.0.0.1:1502:1:50:d1:]", VialPresent_Gpio := 'FC_VialPresent', VialPresent_Modbus := "modbus[127.0.0.1:1502:1:50:d2:]", Stoppered_Gpio := 'FC_Stoppered', Stoppered_Modbus := "modbus[127.0.0.1:1502:1:50:d3:]", Checked_Gpio := 'FC_Checked', Checked_Modbus := "modbus[127.0.0.1:1502:1:50:d4:]", DoorClosed_Gpio := 'FC_DoorClosed', DoorClosed_Modbus := "modbus[127.0.0.1:1502:1:50:d5:]", FilledMl_Gpio := '', FilledMl_Modbus := "modbus[127.0.0.1:1502:1:50:i0:]", Sim_NeedleUp := TRUE, Sim_VialPresent := TRUE, Sim_DoorClosed := TRUE);
        UaFacade : fillingcell::UNIT_Facade(UaRoot := "/Objects/FillingCell/Filler", UaEnable := TRUE);
        Occupation : fillingcell::FC_Occupation;
        Unit : fillingcell::FC_Unit;
        Facade : fillingcell::FC_ProcedureFacade;
      END_FBS
      SUBAPPLICATION EM_Filler (* Equipment module: one composite per skill, chained for status; instances and chain may be changed online while the unit is quiescent *)
        EVENT_INPUT
          INIT;
          UNIT_CTL WITH ControlCode;
          UNIT_STAT WITH UnitRunning, UnitQuiescent, UnitState, Mode, Owner, RemoteAllowed;
          SAMPLE WITH Cell;
          CALL_MoveDown WITH P1_MoveDown, P2_MoveDown, P3_MoveDown, P4_MoveDown;
          CALL_Dose WITH P1_Dose, P2_Dose, P3_Dose, P4_Dose;
          CALL_MoveUp WITH P1_MoveUp, P2_MoveUp, P3_MoveUp, P4_MoveUp;
          CALL_Stopper WITH P1_Stopper, P2_Stopper, P3_Stopper, P4_Stopper;
          CALL_Inspect WITH P1_Inspect, P2_Inspect, P3_Inspect, P4_Inspect;
        END_EVENT
        EVENT_OUTPUT
          INITO;
          STAT_OUT WITH Busy, HeldAll, RunAll;
          DONE_MoveDown;
          DONE_Dose;
          DONE_MoveUp;
          DONE_Stopper;
          DONE_Inspect;
          FAILED_MoveDown WITH CallError_MoveDown;
          FAILED_Dose WITH CallError_Dose;
          FAILED_MoveUp WITH CallError_MoveUp;
          FAILED_Stopper WITH CallError_Stopper;
          FAILED_Inspect WITH CallError_Inspect;
        END_EVENT
        VAR_INPUT
          ControlCode : USINT;
          UnitRunning : BOOL;
          UnitQuiescent : BOOL;
          UnitState : USINT;
          Mode : USINT;
          Owner : UDINT;
          RemoteAllowed : BOOL;
          Cell : fillingcell::ST_CellState;
          P1_MoveDown : LREAL;
          P2_MoveDown : LREAL;
          P3_MoveDown : LREAL;
          P4_MoveDown : LREAL;
          P1_Dose : LREAL;
          P2_Dose : LREAL;
          P3_Dose : LREAL;
          P4_Dose : LREAL;
          P1_MoveUp : LREAL;
          P2_MoveUp : LREAL;
          P3_MoveUp : LREAL;
          P4_MoveUp : LREAL;
          P1_Stopper : LREAL;
          P2_Stopper : LREAL;
          P3_Stopper : LREAL;
          P4_Stopper : LREAL;
          P1_Inspect : LREAL;
          P2_Inspect : LREAL;
          P3_Inspect : LREAL;
          P4_Inspect : LREAL;
        END_VAR
        VAR_OUTPUT
          Busy : BOOL;
          HeldAll : BOOL;
          RunAll : BOOL;
          CallError_MoveDown : UINT;
          CallError_Dose : UINT;
          CallError_MoveUp : UINT;
          CallError_Stopper : UINT;
          CallError_Inspect : UINT;
          Drive_MoveDown : BOOL;
          Drive_Dose : BOOL;
          Drive_MoveUp : BOOL;
          Drive_Stopper : BOOL;
          Drive_Inspect : BOOL;
        END_VAR
        FBS
          MoveDown : fillingcell::SK_MoveDown(UaRoot := "/Objects/FillingCell/Filler/Skills/MoveDown", UaEnable := TRUE, IoBackend := 0, DoGpio := 'FC_MoveDown', DoModbus := "modbus[127.0.0.1:1502:1:0::c0]");
          Dose : fillingcell::SK_Dose(UaRoot := "/Objects/FillingCell/Filler/Skills/Dose", UaEnable := TRUE, IoBackend := 0, DoGpio := 'FC_Dose', DoModbus := "modbus[127.0.0.1:1502:1:0::c1]");
          MoveUp : fillingcell::SK_MoveUp(UaRoot := "/Objects/FillingCell/Filler/Skills/MoveUp", UaEnable := TRUE, IoBackend := 0, DoGpio := 'FC_MoveUp', DoModbus := "modbus[127.0.0.1:1502:1:0::c2]");
          Stopper : fillingcell::SK_Stopper(UaRoot := "/Objects/FillingCell/Filler/Skills/Stopper", UaEnable := TRUE, IoBackend := 0, DoGpio := 'FC_Stopper', DoModbus := "modbus[127.0.0.1:1502:1:0::c3]");
          Inspect : fillingcell::SK_Inspect(UaRoot := "/Objects/FillingCell/Filler/Skills/Inspect", UaEnable := TRUE, IoBackend := 0, DoGpio := 'FC_Inspect', DoModbus := "modbus[127.0.0.1:1502:1:0::c4]");
        END_FBS
        EVENT_CONNECTIONS
          INIT TO MoveDown.INIT;
          MoveDown.INITO TO Dose.INIT;
          MoveDown.STAT_OUT TO Dose.STAT_IN;
          Dose.INITO TO MoveUp.INIT;
          Dose.STAT_OUT TO MoveUp.STAT_IN;
          MoveUp.INITO TO Stopper.INIT;
          MoveUp.STAT_OUT TO Stopper.STAT_IN;
          Stopper.INITO TO Inspect.INIT;
          Stopper.STAT_OUT TO Inspect.STAT_IN;
          Inspect.INITO TO INITO;
          Inspect.STAT_OUT TO STAT_OUT;
          UNIT_CTL TO MoveDown.UNIT_CTL;
          UNIT_STAT TO MoveDown.UNIT_STAT;
          SAMPLE TO MoveDown.SAMPLE;
          CALL_MoveDown TO MoveDown.CALL;
          MoveDown.DONE TO DONE_MoveDown;
          MoveDown.FAILED TO FAILED_MoveDown;
          UNIT_CTL TO Dose.UNIT_CTL;
          UNIT_STAT TO Dose.UNIT_STAT;
          SAMPLE TO Dose.SAMPLE;
          CALL_Dose TO Dose.CALL;
          Dose.DONE TO DONE_Dose;
          Dose.FAILED TO FAILED_Dose;
          UNIT_CTL TO MoveUp.UNIT_CTL;
          UNIT_STAT TO MoveUp.UNIT_STAT;
          SAMPLE TO MoveUp.SAMPLE;
          CALL_MoveUp TO MoveUp.CALL;
          MoveUp.DONE TO DONE_MoveUp;
          MoveUp.FAILED TO FAILED_MoveUp;
          UNIT_CTL TO Stopper.UNIT_CTL;
          UNIT_STAT TO Stopper.UNIT_STAT;
          SAMPLE TO Stopper.SAMPLE;
          CALL_Stopper TO Stopper.CALL;
          Stopper.DONE TO DONE_Stopper;
          Stopper.FAILED TO FAILED_Stopper;
          UNIT_CTL TO Inspect.UNIT_CTL;
          UNIT_STAT TO Inspect.UNIT_STAT;
          SAMPLE TO Inspect.SAMPLE;
          CALL_Inspect TO Inspect.CALL;
          Inspect.DONE TO DONE_Inspect;
          Inspect.FAILED TO FAILED_Inspect;
        END_CONNECTIONS
        DATA_CONNECTIONS
          MoveDown.BusyOut TO Dose.BusyIn;
          MoveDown.HeldOut TO Dose.HeldIn;
          MoveDown.RunOut TO Dose.RunIn;
          Dose.BusyOut TO MoveUp.BusyIn;
          Dose.HeldOut TO MoveUp.HeldIn;
          Dose.RunOut TO MoveUp.RunIn;
          MoveUp.BusyOut TO Stopper.BusyIn;
          MoveUp.HeldOut TO Stopper.HeldIn;
          MoveUp.RunOut TO Stopper.RunIn;
          Stopper.BusyOut TO Inspect.BusyIn;
          Stopper.HeldOut TO Inspect.HeldIn;
          Stopper.RunOut TO Inspect.RunIn;
          Inspect.BusyOut TO Busy;
          Inspect.HeldOut TO HeldAll;
          Inspect.RunOut TO RunAll;
          ControlCode TO MoveDown.ControlCode;
          Cell TO MoveDown.Cell;
          MoveDown.CallError TO CallError_MoveDown;
          MoveDown.Drive TO Drive_MoveDown;
          UnitRunning TO MoveDown.UnitRunning;
          UnitQuiescent TO MoveDown.UnitQuiescent;
          UnitState TO MoveDown.UnitState;
          Mode TO MoveDown.Mode;
          Owner TO MoveDown.Owner;
          RemoteAllowed TO MoveDown.RemoteAllowed;
          P1_MoveDown TO MoveDown.P1;
          P2_MoveDown TO MoveDown.P2;
          P3_MoveDown TO MoveDown.P3;
          P4_MoveDown TO MoveDown.P4;
          ControlCode TO Dose.ControlCode;
          Cell TO Dose.Cell;
          Dose.CallError TO CallError_Dose;
          Dose.Drive TO Drive_Dose;
          UnitRunning TO Dose.UnitRunning;
          UnitQuiescent TO Dose.UnitQuiescent;
          UnitState TO Dose.UnitState;
          Mode TO Dose.Mode;
          Owner TO Dose.Owner;
          RemoteAllowed TO Dose.RemoteAllowed;
          P1_Dose TO Dose.P1;
          P2_Dose TO Dose.P2;
          P3_Dose TO Dose.P3;
          P4_Dose TO Dose.P4;
          ControlCode TO MoveUp.ControlCode;
          Cell TO MoveUp.Cell;
          MoveUp.CallError TO CallError_MoveUp;
          MoveUp.Drive TO Drive_MoveUp;
          UnitRunning TO MoveUp.UnitRunning;
          UnitQuiescent TO MoveUp.UnitQuiescent;
          UnitState TO MoveUp.UnitState;
          Mode TO MoveUp.Mode;
          Owner TO MoveUp.Owner;
          RemoteAllowed TO MoveUp.RemoteAllowed;
          P1_MoveUp TO MoveUp.P1;
          P2_MoveUp TO MoveUp.P2;
          P3_MoveUp TO MoveUp.P3;
          P4_MoveUp TO MoveUp.P4;
          ControlCode TO Stopper.ControlCode;
          Cell TO Stopper.Cell;
          Stopper.CallError TO CallError_Stopper;
          Stopper.Drive TO Drive_Stopper;
          UnitRunning TO Stopper.UnitRunning;
          UnitQuiescent TO Stopper.UnitQuiescent;
          UnitState TO Stopper.UnitState;
          Mode TO Stopper.Mode;
          Owner TO Stopper.Owner;
          RemoteAllowed TO Stopper.RemoteAllowed;
          P1_Stopper TO Stopper.P1;
          P2_Stopper TO Stopper.P2;
          P3_Stopper TO Stopper.P3;
          P4_Stopper TO Stopper.P4;
          ControlCode TO Inspect.ControlCode;
          Cell TO Inspect.Cell;
          Inspect.CallError TO CallError_Inspect;
          Inspect.Drive TO Drive_Inspect;
          UnitRunning TO Inspect.UnitRunning;
          UnitQuiescent TO Inspect.UnitQuiescent;
          UnitState TO Inspect.UnitState;
          Mode TO Inspect.Mode;
          Owner TO Inspect.Owner;
          RemoteAllowed TO Inspect.RemoteAllowed;
          P1_Inspect TO Inspect.P1;
          P2_Inspect TO Inspect.P2;
          P3_Inspect TO Inspect.P3;
          P4_Inspect TO Inspect.P4;
        END_CONNECTIONS
      END_SUBAPPLICATION
      SUBAPPLICATION PROC (* INTENTIONALLY EMPTY: generated procedure (P_* pattern instances) calls skills via CALL_*/DONE_*/FAILED_* *)
        EVENT_INPUT
          START;
          RESET;
          CMD WITH Command;
          DONE_MoveDown;
          DONE_Dose;
          DONE_MoveUp;
          DONE_Stopper;
          DONE_Inspect;
          FAILED_MoveDown WITH CallError_MoveDown;
          FAILED_Dose WITH CallError_Dose;
          FAILED_MoveUp WITH CallError_MoveUp;
          FAILED_Stopper WITH CallError_Stopper;
          FAILED_Inspect WITH CallError_Inspect;
        END_EVENT
        EVENT_OUTPUT
          FINISHED;
          FAILED;
          CALL_MoveDown WITH P1_MoveDown, P2_MoveDown, P3_MoveDown, P4_MoveDown;
          CALL_Dose WITH P1_Dose, P2_Dose, P3_Dose, P4_Dose;
          CALL_MoveUp WITH P1_MoveUp, P2_MoveUp, P3_MoveUp, P4_MoveUp;
          CALL_Stopper WITH P1_Stopper, P2_Stopper, P3_Stopper, P4_Stopper;
          CALL_Inspect WITH P1_Inspect, P2_Inspect, P3_Inspect, P4_Inspect;
        END_EVENT
        VAR_INPUT
          Command : USINT;
          CallError_MoveDown : UINT;
          CallError_Dose : UINT;
          CallError_MoveUp : UINT;
          CallError_Stopper : UINT;
          CallError_Inspect : UINT;
        END_VAR
        VAR_OUTPUT
          P1_MoveDown : LREAL;
          P2_MoveDown : LREAL;
          P3_MoveDown : LREAL;
          P4_MoveDown : LREAL;
          P1_Dose : LREAL;
          P2_Dose : LREAL;
          P3_Dose : LREAL;
          P4_Dose : LREAL;
          P1_MoveUp : LREAL;
          P2_MoveUp : LREAL;
          P3_MoveUp : LREAL;
          P4_MoveUp : LREAL;
          P1_Stopper : LREAL;
          P2_Stopper : LREAL;
          P3_Stopper : LREAL;
          P4_Stopper : LREAL;
          P1_Inspect : LREAL;
          P2_Inspect : LREAL;
          P3_Inspect : LREAL;
          P4_Inspect : LREAL;
        END_VAR
      END_SUBAPPLICATION
      EVENT_CONNECTIONS
        Boot.COLD TO Observer.INIT;
        Boot.WARM TO Observer.INIT;
        Unit.CNF TO EM_Filler.UNIT_STAT;
        Occupation.CNF TO EM_Filler.UNIT_STAT;
        Unit.CONTROL TO EM_Filler.UNIT_CTL;
        EM_Filler.STAT_OUT TO Unit.STATUS;
        Observer.SAMPLE TO EM_Filler.SAMPLE;
        Observer.UNSAFE TO Unit.UNSAFE;
        Unit.PROC_CMD TO Facade.CMD;
        Facade.EXEC TO PROC.CMD;
        Facade.START TO PROC.START;
        Facade.RESET TO PROC.RESET;
        PROC.FINISHED TO Facade.FINISHED;
        PROC.FAILED TO Facade.FAILED;
        Facade.DONE TO Unit.PROC_DONE;
        Facade.FAULT TO Unit.FAULT;
        PROC.CALL_MoveDown TO EM_Filler.CALL_MoveDown;
        EM_Filler.DONE_MoveDown TO PROC.DONE_MoveDown;
        EM_Filler.FAILED_MoveDown TO PROC.FAILED_MoveDown;
        PROC.CALL_Dose TO EM_Filler.CALL_Dose;
        EM_Filler.DONE_Dose TO PROC.DONE_Dose;
        EM_Filler.FAILED_Dose TO PROC.FAILED_Dose;
        PROC.CALL_MoveUp TO EM_Filler.CALL_MoveUp;
        EM_Filler.DONE_MoveUp TO PROC.DONE_MoveUp;
        EM_Filler.FAILED_MoveUp TO PROC.FAILED_MoveUp;
        PROC.CALL_Stopper TO EM_Filler.CALL_Stopper;
        EM_Filler.DONE_Stopper TO PROC.DONE_Stopper;
        EM_Filler.FAILED_Stopper TO PROC.FAILED_Stopper;
        PROC.CALL_Inspect TO EM_Filler.CALL_Inspect;
        EM_Filler.DONE_Inspect TO PROC.DONE_Inspect;
        EM_Filler.FAILED_Inspect TO PROC.FAILED_Inspect;
        Observer.INITO TO UaFacade.INIT;
        UaFacade.INITO TO EM_Filler.INIT;
        UaFacade.U_CMD TO Unit.CMD;
        UaFacade.O_CMD TO Occupation.CMD;
        Unit.CMD_ACK TO UaFacade.U_ACK;
        Unit.CMD_REJ TO UaFacade.U_REJ;
        Occupation.CNF TO UaFacade.O_ACK;
        Occupation.REJECTED TO UaFacade.O_REJ;
        Unit.CNF TO UaFacade.PUB;
        Occupation.CNF TO UaFacade.PUB;
      END_CONNECTIONS
      DATA_CONNECTIONS
        Occupation.Owner TO Unit.Owner;
        Occupation.RemoteAllowed TO Unit.RemoteAllowed;
        Occupation.Owner TO EM_Filler.Owner;
        Occupation.RemoteAllowed TO EM_Filler.RemoteAllowed;
        Unit.Running TO EM_Filler.UnitRunning;
        Unit.Quiescent TO EM_Filler.UnitQuiescent;
        Unit.State TO EM_Filler.UnitState;
        Unit.Mode TO EM_Filler.Mode;
        Unit.ControlCode TO EM_Filler.ControlCode;
        Unit.Quiescent TO Occupation.Quiescent;
        Unit.Quiescent TO Facade.Quiescent;
        EM_Filler.Busy TO Unit.Busy;
        EM_Filler.HeldAll TO Unit.HeldAll;
        EM_Filler.RunAll TO Unit.RunAll;
        Observer.Cell TO EM_Filler.Cell;
        Observer.Safe TO Unit.Safe;
        Unit.ProcedureCommand TO Facade.Command;
        Facade.CommandOut TO PROC.Command;
        Facade.Ready TO Unit.ProcedureReady;
        PROC.P1_MoveDown TO EM_Filler.P1_MoveDown;
        PROC.P2_MoveDown TO EM_Filler.P2_MoveDown;
        PROC.P3_MoveDown TO EM_Filler.P3_MoveDown;
        PROC.P4_MoveDown TO EM_Filler.P4_MoveDown;
        EM_Filler.CallError_MoveDown TO PROC.CallError_MoveDown;
        PROC.P1_Dose TO EM_Filler.P1_Dose;
        PROC.P2_Dose TO EM_Filler.P2_Dose;
        PROC.P3_Dose TO EM_Filler.P3_Dose;
        PROC.P4_Dose TO EM_Filler.P4_Dose;
        EM_Filler.CallError_Dose TO PROC.CallError_Dose;
        PROC.P1_MoveUp TO EM_Filler.P1_MoveUp;
        PROC.P2_MoveUp TO EM_Filler.P2_MoveUp;
        PROC.P3_MoveUp TO EM_Filler.P3_MoveUp;
        PROC.P4_MoveUp TO EM_Filler.P4_MoveUp;
        EM_Filler.CallError_MoveUp TO PROC.CallError_MoveUp;
        PROC.P1_Stopper TO EM_Filler.P1_Stopper;
        PROC.P2_Stopper TO EM_Filler.P2_Stopper;
        PROC.P3_Stopper TO EM_Filler.P3_Stopper;
        PROC.P4_Stopper TO EM_Filler.P4_Stopper;
        EM_Filler.CallError_Stopper TO PROC.CallError_Stopper;
        PROC.P1_Inspect TO EM_Filler.P1_Inspect;
        PROC.P2_Inspect TO EM_Filler.P2_Inspect;
        PROC.P3_Inspect TO EM_Filler.P3_Inspect;
        PROC.P4_Inspect TO EM_Filler.P4_Inspect;
        EM_Filler.CallError_Inspect TO PROC.CallError_Inspect;
        UaFacade.Requester TO Unit.Requester;
        UaFacade.Requester TO Occupation.Requester;
        UaFacade.U_Code TO Unit.Command;
        UaFacade.U_Mode TO Unit.RequestedMode;
        UaFacade.O_Code TO Occupation.Command;
        Unit.State TO UaFacade.UnitState;
        Unit.Mode TO UaFacade.UnitMode;
        Occupation.State TO UaFacade.OccState;
        Occupation.Owner TO UaFacade.Owner;
      END_CONNECTIONS
    END_RESOURCE
    RESOURCE DEMO : iec61499::system::EMB_RES
      FBS
        Boot : iec61499::events::E_RESTART;
        Observer : fillingcell::UNIT_Observer(UaRoot := "/Objects/Demo/Filler", UaEnable := FALSE, IoBackend := 0, CycleTime := T#50ms);
        Occupation : fillingcell::FC_Occupation;
        Unit : fillingcell::FC_Unit;
        Facade : fillingcell::FC_ProcedureFacade(Installed := TRUE);
        Plant : fillingcell::DEMO_Plant;
        PlantClock : iec61499::events::E_CYCLE(DT := T#20ms);
        Operator : fillingcell::DEMO_Operator;
        OpDelay : iec61499::events::E_DELAY;
      END_FBS
      SUBAPPLICATION EM_Filler (* Equipment module: one composite per skill, chained for status; instances and chain may be changed online while the unit is quiescent *)
        EVENT_INPUT
          INIT;
          UNIT_CTL WITH ControlCode;
          UNIT_STAT WITH UnitRunning, UnitQuiescent, UnitState, Mode, Owner, RemoteAllowed;
          SAMPLE WITH Cell;
          CALL_MoveDown WITH P1_MoveDown, P2_MoveDown, P3_MoveDown, P4_MoveDown;
          CALL_Dose WITH P1_Dose, P2_Dose, P3_Dose, P4_Dose;
          CALL_MoveUp WITH P1_MoveUp, P2_MoveUp, P3_MoveUp, P4_MoveUp;
          CALL_Stopper WITH P1_Stopper, P2_Stopper, P3_Stopper, P4_Stopper;
          CALL_Inspect WITH P1_Inspect, P2_Inspect, P3_Inspect, P4_Inspect;
        END_EVENT
        EVENT_OUTPUT
          INITO;
          STAT_OUT WITH Busy, HeldAll, RunAll;
          DONE_MoveDown;
          DONE_Dose;
          DONE_MoveUp;
          DONE_Stopper;
          DONE_Inspect;
          FAILED_MoveDown WITH CallError_MoveDown;
          FAILED_Dose WITH CallError_Dose;
          FAILED_MoveUp WITH CallError_MoveUp;
          FAILED_Stopper WITH CallError_Stopper;
          FAILED_Inspect WITH CallError_Inspect;
        END_EVENT
        VAR_INPUT
          ControlCode : USINT;
          UnitRunning : BOOL;
          UnitQuiescent : BOOL;
          UnitState : USINT;
          Mode : USINT;
          Owner : UDINT;
          RemoteAllowed : BOOL;
          Cell : fillingcell::ST_CellState;
          P1_MoveDown : LREAL;
          P2_MoveDown : LREAL;
          P3_MoveDown : LREAL;
          P4_MoveDown : LREAL;
          P1_Dose : LREAL;
          P2_Dose : LREAL;
          P3_Dose : LREAL;
          P4_Dose : LREAL;
          P1_MoveUp : LREAL;
          P2_MoveUp : LREAL;
          P3_MoveUp : LREAL;
          P4_MoveUp : LREAL;
          P1_Stopper : LREAL;
          P2_Stopper : LREAL;
          P3_Stopper : LREAL;
          P4_Stopper : LREAL;
          P1_Inspect : LREAL;
          P2_Inspect : LREAL;
          P3_Inspect : LREAL;
          P4_Inspect : LREAL;
        END_VAR
        VAR_OUTPUT
          Busy : BOOL;
          HeldAll : BOOL;
          RunAll : BOOL;
          CallError_MoveDown : UINT;
          CallError_Dose : UINT;
          CallError_MoveUp : UINT;
          CallError_Stopper : UINT;
          CallError_Inspect : UINT;
          Drive_MoveDown : BOOL;
          Drive_Dose : BOOL;
          Drive_MoveUp : BOOL;
          Drive_Stopper : BOOL;
          Drive_Inspect : BOOL;
        END_VAR
        FBS
          MoveDown : fillingcell::SK_MoveDown(UaRoot := "/Objects/Demo/Filler/Skills/MoveDown", UaEnable := FALSE, IoBackend := 0);
          Dose : fillingcell::SK_Dose(UaRoot := "/Objects/Demo/Filler/Skills/Dose", UaEnable := FALSE, IoBackend := 0);
          MoveUp : fillingcell::SK_MoveUp(UaRoot := "/Objects/Demo/Filler/Skills/MoveUp", UaEnable := FALSE, IoBackend := 0);
          Stopper : fillingcell::SK_Stopper(UaRoot := "/Objects/Demo/Filler/Skills/Stopper", UaEnable := FALSE, IoBackend := 0);
          Inspect : fillingcell::SK_Inspect(UaRoot := "/Objects/Demo/Filler/Skills/Inspect", UaEnable := FALSE, IoBackend := 0);
        END_FBS
        EVENT_CONNECTIONS
          INIT TO MoveDown.INIT;
          MoveDown.INITO TO Dose.INIT;
          MoveDown.STAT_OUT TO Dose.STAT_IN;
          Dose.INITO TO MoveUp.INIT;
          Dose.STAT_OUT TO MoveUp.STAT_IN;
          MoveUp.INITO TO Stopper.INIT;
          MoveUp.STAT_OUT TO Stopper.STAT_IN;
          Stopper.INITO TO Inspect.INIT;
          Stopper.STAT_OUT TO Inspect.STAT_IN;
          Inspect.INITO TO INITO;
          Inspect.STAT_OUT TO STAT_OUT;
          UNIT_CTL TO MoveDown.UNIT_CTL;
          UNIT_STAT TO MoveDown.UNIT_STAT;
          SAMPLE TO MoveDown.SAMPLE;
          CALL_MoveDown TO MoveDown.CALL;
          MoveDown.DONE TO DONE_MoveDown;
          MoveDown.FAILED TO FAILED_MoveDown;
          UNIT_CTL TO Dose.UNIT_CTL;
          UNIT_STAT TO Dose.UNIT_STAT;
          SAMPLE TO Dose.SAMPLE;
          CALL_Dose TO Dose.CALL;
          Dose.DONE TO DONE_Dose;
          Dose.FAILED TO FAILED_Dose;
          UNIT_CTL TO MoveUp.UNIT_CTL;
          UNIT_STAT TO MoveUp.UNIT_STAT;
          SAMPLE TO MoveUp.SAMPLE;
          CALL_MoveUp TO MoveUp.CALL;
          MoveUp.DONE TO DONE_MoveUp;
          MoveUp.FAILED TO FAILED_MoveUp;
          UNIT_CTL TO Stopper.UNIT_CTL;
          UNIT_STAT TO Stopper.UNIT_STAT;
          SAMPLE TO Stopper.SAMPLE;
          CALL_Stopper TO Stopper.CALL;
          Stopper.DONE TO DONE_Stopper;
          Stopper.FAILED TO FAILED_Stopper;
          UNIT_CTL TO Inspect.UNIT_CTL;
          UNIT_STAT TO Inspect.UNIT_STAT;
          SAMPLE TO Inspect.SAMPLE;
          CALL_Inspect TO Inspect.CALL;
          Inspect.DONE TO DONE_Inspect;
          Inspect.FAILED TO FAILED_Inspect;
        END_CONNECTIONS
        DATA_CONNECTIONS
          MoveDown.BusyOut TO Dose.BusyIn;
          MoveDown.HeldOut TO Dose.HeldIn;
          MoveDown.RunOut TO Dose.RunIn;
          Dose.BusyOut TO MoveUp.BusyIn;
          Dose.HeldOut TO MoveUp.HeldIn;
          Dose.RunOut TO MoveUp.RunIn;
          MoveUp.BusyOut TO Stopper.BusyIn;
          MoveUp.HeldOut TO Stopper.HeldIn;
          MoveUp.RunOut TO Stopper.RunIn;
          Stopper.BusyOut TO Inspect.BusyIn;
          Stopper.HeldOut TO Inspect.HeldIn;
          Stopper.RunOut TO Inspect.RunIn;
          Inspect.BusyOut TO Busy;
          Inspect.HeldOut TO HeldAll;
          Inspect.RunOut TO RunAll;
          ControlCode TO MoveDown.ControlCode;
          Cell TO MoveDown.Cell;
          MoveDown.CallError TO CallError_MoveDown;
          MoveDown.Drive TO Drive_MoveDown;
          UnitRunning TO MoveDown.UnitRunning;
          UnitQuiescent TO MoveDown.UnitQuiescent;
          UnitState TO MoveDown.UnitState;
          Mode TO MoveDown.Mode;
          Owner TO MoveDown.Owner;
          RemoteAllowed TO MoveDown.RemoteAllowed;
          P1_MoveDown TO MoveDown.P1;
          P2_MoveDown TO MoveDown.P2;
          P3_MoveDown TO MoveDown.P3;
          P4_MoveDown TO MoveDown.P4;
          ControlCode TO Dose.ControlCode;
          Cell TO Dose.Cell;
          Dose.CallError TO CallError_Dose;
          Dose.Drive TO Drive_Dose;
          UnitRunning TO Dose.UnitRunning;
          UnitQuiescent TO Dose.UnitQuiescent;
          UnitState TO Dose.UnitState;
          Mode TO Dose.Mode;
          Owner TO Dose.Owner;
          RemoteAllowed TO Dose.RemoteAllowed;
          P1_Dose TO Dose.P1;
          P2_Dose TO Dose.P2;
          P3_Dose TO Dose.P3;
          P4_Dose TO Dose.P4;
          ControlCode TO MoveUp.ControlCode;
          Cell TO MoveUp.Cell;
          MoveUp.CallError TO CallError_MoveUp;
          MoveUp.Drive TO Drive_MoveUp;
          UnitRunning TO MoveUp.UnitRunning;
          UnitQuiescent TO MoveUp.UnitQuiescent;
          UnitState TO MoveUp.UnitState;
          Mode TO MoveUp.Mode;
          Owner TO MoveUp.Owner;
          RemoteAllowed TO MoveUp.RemoteAllowed;
          P1_MoveUp TO MoveUp.P1;
          P2_MoveUp TO MoveUp.P2;
          P3_MoveUp TO MoveUp.P3;
          P4_MoveUp TO MoveUp.P4;
          ControlCode TO Stopper.ControlCode;
          Cell TO Stopper.Cell;
          Stopper.CallError TO CallError_Stopper;
          Stopper.Drive TO Drive_Stopper;
          UnitRunning TO Stopper.UnitRunning;
          UnitQuiescent TO Stopper.UnitQuiescent;
          UnitState TO Stopper.UnitState;
          Mode TO Stopper.Mode;
          Owner TO Stopper.Owner;
          RemoteAllowed TO Stopper.RemoteAllowed;
          P1_Stopper TO Stopper.P1;
          P2_Stopper TO Stopper.P2;
          P3_Stopper TO Stopper.P3;
          P4_Stopper TO Stopper.P4;
          ControlCode TO Inspect.ControlCode;
          Cell TO Inspect.Cell;
          Inspect.CallError TO CallError_Inspect;
          Inspect.Drive TO Drive_Inspect;
          UnitRunning TO Inspect.UnitRunning;
          UnitQuiescent TO Inspect.UnitQuiescent;
          UnitState TO Inspect.UnitState;
          Mode TO Inspect.Mode;
          Owner TO Inspect.Owner;
          RemoteAllowed TO Inspect.RemoteAllowed;
          P1_Inspect TO Inspect.P1;
          P2_Inspect TO Inspect.P2;
          P3_Inspect TO Inspect.P3;
          P4_Inspect TO Inspect.P4;
        END_CONNECTIONS
      END_SUBAPPLICATION
      SUBAPPLICATION PROC (* Demo procedure: MoveDown, Dose x2 (P_Loop), MoveUp, Stopper, Inspect *)
        EVENT_INPUT
          START;
          RESET;
          CMD WITH Command;
          DONE_MoveDown;
          DONE_Dose;
          DONE_MoveUp;
          DONE_Stopper;
          DONE_Inspect;
          FAILED_MoveDown WITH CallError_MoveDown;
          FAILED_Dose WITH CallError_Dose;
          FAILED_MoveUp WITH CallError_MoveUp;
          FAILED_Stopper WITH CallError_Stopper;
          FAILED_Inspect WITH CallError_Inspect;
        END_EVENT
        EVENT_OUTPUT
          FINISHED;
          FAILED;
          CALL_MoveDown WITH P1_MoveDown, P2_MoveDown, P3_MoveDown, P4_MoveDown;
          CALL_Dose WITH P1_Dose, P2_Dose, P3_Dose, P4_Dose;
          CALL_MoveUp WITH P1_MoveUp, P2_MoveUp, P3_MoveUp, P4_MoveUp;
          CALL_Stopper WITH P1_Stopper, P2_Stopper, P3_Stopper, P4_Stopper;
          CALL_Inspect WITH P1_Inspect, P2_Inspect, P3_Inspect, P4_Inspect;
        END_EVENT
        VAR_INPUT
          Command : USINT;
          CallError_MoveDown : UINT;
          CallError_Dose : UINT;
          CallError_MoveUp : UINT;
          CallError_Stopper : UINT;
          CallError_Inspect : UINT;
        END_VAR
        VAR_OUTPUT
          P1_MoveDown : LREAL;
          P2_MoveDown : LREAL;
          P3_MoveDown : LREAL;
          P4_MoveDown : LREAL;
          P1_Dose : LREAL;
          P2_Dose : LREAL;
          P3_Dose : LREAL;
          P4_Dose : LREAL;
          P1_MoveUp : LREAL;
          P2_MoveUp : LREAL;
          P3_MoveUp : LREAL;
          P4_MoveUp : LREAL;
          P1_Stopper : LREAL;
          P2_Stopper : LREAL;
          P3_Stopper : LREAL;
          P4_Stopper : LREAL;
          P1_Inspect : LREAL;
          P2_Inspect : LREAL;
          P3_Inspect : LREAL;
          P4_Inspect : LREAL;
        END_VAR
        FBS
          MoveDown : fillingcell::P_Call;
          Dose : fillingcell::P_Call(P1 := 0.3);
          MoveUp : fillingcell::P_Call;
          Stopper : fillingcell::P_Call;
          Inspect : fillingcell::P_Call;
          DoseLoop : fillingcell::P_Loop(Count := 2);
        END_FBS
        EVENT_CONNECTIONS
          START TO MoveDown.EI;
          MoveDown.EO TO DoseLoop.EI;
          DoseLoop.BODY TO Dose.EI;
          Dose.EO TO DoseLoop.NEXT;
          DoseLoop.EO TO MoveUp.EI;
          MoveUp.EO TO Stopper.EI;
          Stopper.EO TO Inspect.EI;
          Inspect.EO TO FINISHED;
          RESET TO DoseLoop.RESET;
          MoveDown.CALL TO CALL_MoveDown;
          DONE_MoveDown TO MoveDown.DONE;
          FAILED_MoveDown TO MoveDown.FAILED;
          MoveDown.ERR TO FAILED;
          RESET TO MoveDown.RESET;
          Dose.CALL TO CALL_Dose;
          DONE_Dose TO Dose.DONE;
          FAILED_Dose TO Dose.FAILED;
          Dose.ERR TO FAILED;
          RESET TO Dose.RESET;
          MoveUp.CALL TO CALL_MoveUp;
          DONE_MoveUp TO MoveUp.DONE;
          FAILED_MoveUp TO MoveUp.FAILED;
          MoveUp.ERR TO FAILED;
          RESET TO MoveUp.RESET;
          Stopper.CALL TO CALL_Stopper;
          DONE_Stopper TO Stopper.DONE;
          FAILED_Stopper TO Stopper.FAILED;
          Stopper.ERR TO FAILED;
          RESET TO Stopper.RESET;
          Inspect.CALL TO CALL_Inspect;
          DONE_Inspect TO Inspect.DONE;
          FAILED_Inspect TO Inspect.FAILED;
          Inspect.ERR TO FAILED;
          RESET TO Inspect.RESET;
        END_CONNECTIONS
        DATA_CONNECTIONS
          Dose.CP1 TO P1_Dose;
          CallError_MoveDown TO MoveDown.CallError;
          CallError_Dose TO Dose.CallError;
          CallError_MoveUp TO MoveUp.CallError;
          CallError_Stopper TO Stopper.CallError;
          CallError_Inspect TO Inspect.CallError;
        END_CONNECTIONS
      END_SUBAPPLICATION
      EVENT_CONNECTIONS
        Boot.COLD TO Observer.INIT;
        Boot.WARM TO Observer.INIT;
        Unit.CNF TO EM_Filler.UNIT_STAT;
        Occupation.CNF TO EM_Filler.UNIT_STAT;
        Unit.CONTROL TO EM_Filler.UNIT_CTL;
        EM_Filler.STAT_OUT TO Unit.STATUS;
        Observer.SAMPLE TO EM_Filler.SAMPLE;
        Observer.UNSAFE TO Unit.UNSAFE;
        Unit.PROC_CMD TO Facade.CMD;
        Facade.EXEC TO PROC.CMD;
        Facade.START TO PROC.START;
        Facade.RESET TO PROC.RESET;
        PROC.FINISHED TO Facade.FINISHED;
        PROC.FAILED TO Facade.FAILED;
        Facade.DONE TO Unit.PROC_DONE;
        Facade.FAULT TO Unit.FAULT;
        PROC.CALL_MoveDown TO EM_Filler.CALL_MoveDown;
        EM_Filler.DONE_MoveDown TO PROC.DONE_MoveDown;
        EM_Filler.FAILED_MoveDown TO PROC.FAILED_MoveDown;
        PROC.CALL_Dose TO EM_Filler.CALL_Dose;
        EM_Filler.DONE_Dose TO PROC.DONE_Dose;
        EM_Filler.FAILED_Dose TO PROC.FAILED_Dose;
        PROC.CALL_MoveUp TO EM_Filler.CALL_MoveUp;
        EM_Filler.DONE_MoveUp TO PROC.DONE_MoveUp;
        EM_Filler.FAILED_MoveUp TO PROC.FAILED_MoveUp;
        PROC.CALL_Stopper TO EM_Filler.CALL_Stopper;
        EM_Filler.DONE_Stopper TO PROC.DONE_Stopper;
        EM_Filler.FAILED_Stopper TO PROC.FAILED_Stopper;
        PROC.CALL_Inspect TO EM_Filler.CALL_Inspect;
        EM_Filler.DONE_Inspect TO PROC.DONE_Inspect;
        EM_Filler.FAILED_Inspect TO PROC.FAILED_Inspect;
        Boot.COLD TO Plant.INIT;
        Boot.WARM TO Plant.INIT;
        Boot.COLD TO PlantClock.START;
        Boot.WARM TO PlantClock.START;
        PlantClock.EO TO Plant.TICK;
        Plant.CNF TO Observer.SIM;
        Observer.INITO TO EM_Filler.INIT;
        EM_Filler.INITO TO Facade.CONFIG;
        Facade.CNF TO Operator.START;
        Operator.O_CMD TO Occupation.CMD;
        Operator.U_CMD TO Unit.CMD;
        Operator.NEW_VIAL TO Plant.NEW_VIAL;
        Operator.WAIT TO OpDelay.START;
        OpDelay.EO TO Operator.TIMER;
        Unit.CNF TO Operator.UNIT;
        Unit.CMD_REJ TO Operator.REJ;
      END_CONNECTIONS
      DATA_CONNECTIONS
        Occupation.Owner TO Unit.Owner;
        Occupation.RemoteAllowed TO Unit.RemoteAllowed;
        Occupation.Owner TO EM_Filler.Owner;
        Occupation.RemoteAllowed TO EM_Filler.RemoteAllowed;
        Unit.Running TO EM_Filler.UnitRunning;
        Unit.Quiescent TO EM_Filler.UnitQuiescent;
        Unit.State TO EM_Filler.UnitState;
        Unit.Mode TO EM_Filler.Mode;
        Unit.ControlCode TO EM_Filler.ControlCode;
        Unit.Quiescent TO Occupation.Quiescent;
        Unit.Quiescent TO Facade.Quiescent;
        EM_Filler.Busy TO Unit.Busy;
        EM_Filler.HeldAll TO Unit.HeldAll;
        EM_Filler.RunAll TO Unit.RunAll;
        Observer.Cell TO EM_Filler.Cell;
        Observer.Safe TO Unit.Safe;
        Unit.ProcedureCommand TO Facade.Command;
        Facade.CommandOut TO PROC.Command;
        Facade.Ready TO Unit.ProcedureReady;
        PROC.P1_MoveDown TO EM_Filler.P1_MoveDown;
        PROC.P2_MoveDown TO EM_Filler.P2_MoveDown;
        PROC.P3_MoveDown TO EM_Filler.P3_MoveDown;
        PROC.P4_MoveDown TO EM_Filler.P4_MoveDown;
        EM_Filler.CallError_MoveDown TO PROC.CallError_MoveDown;
        PROC.P1_Dose TO EM_Filler.P1_Dose;
        PROC.P2_Dose TO EM_Filler.P2_Dose;
        PROC.P3_Dose TO EM_Filler.P3_Dose;
        PROC.P4_Dose TO EM_Filler.P4_Dose;
        EM_Filler.CallError_Dose TO PROC.CallError_Dose;
        PROC.P1_MoveUp TO EM_Filler.P1_MoveUp;
        PROC.P2_MoveUp TO EM_Filler.P2_MoveUp;
        PROC.P3_MoveUp TO EM_Filler.P3_MoveUp;
        PROC.P4_MoveUp TO EM_Filler.P4_MoveUp;
        EM_Filler.CallError_MoveUp TO PROC.CallError_MoveUp;
        PROC.P1_Stopper TO EM_Filler.P1_Stopper;
        PROC.P2_Stopper TO EM_Filler.P2_Stopper;
        PROC.P3_Stopper TO EM_Filler.P3_Stopper;
        PROC.P4_Stopper TO EM_Filler.P4_Stopper;
        EM_Filler.CallError_Stopper TO PROC.CallError_Stopper;
        PROC.P1_Inspect TO EM_Filler.P1_Inspect;
        PROC.P2_Inspect TO EM_Filler.P2_Inspect;
        PROC.P3_Inspect TO EM_Filler.P3_Inspect;
        PROC.P4_Inspect TO EM_Filler.P4_Inspect;
        EM_Filler.CallError_Inspect TO PROC.CallError_Inspect;
        Operator.Requester TO Unit.Requester;
        Operator.Requester TO Occupation.Requester;
        Operator.U_Code TO Unit.Command;
        Operator.U_Mode TO Unit.RequestedMode;
        Operator.O_Code TO Occupation.Command;
        Unit.State TO Operator.UnitState;
        Operator.Delay TO OpDelay.DT;
        Plant.NeedleUp TO Observer.Sim_NeedleUp;
        Plant.NeedleDown TO Observer.Sim_NeedleDown;
        Plant.VialPresent TO Observer.Sim_VialPresent;
        Plant.FilledMl TO Observer.Sim_FilledMl;
        Plant.Stoppered TO Observer.Sim_Stoppered;
        Plant.Checked TO Observer.Sim_Checked;
        Plant.DoorClosed TO Observer.Sim_DoorClosed;
        EM_Filler.Drive_MoveDown TO Plant.DriveMoveDown;
        EM_Filler.Drive_Dose TO Plant.DriveDose;
        EM_Filler.Drive_MoveUp TO Plant.DriveMoveUp;
        EM_Filler.Drive_Stopper TO Plant.DriveStopper;
        EM_Filler.Drive_Inspect TO Plant.DriveInspect;
      END_CONNECTIONS
    END_RESOURCE
    RESOURCE BENCH : iec61499::system::EMB_RES
      FBS
        Boot : iec61499::events::E_RESTART;
        Plant : fillingcell::DEMO_Plant(StartDown := TRUE);
        PlantClock : iec61499::events::E_CYCLE(DT := T#20ms);
        Observer : fillingcell::UNIT_Observer(UaRoot := "/Objects/Demo/Bench", UaEnable := FALSE, IoBackend := 0, CycleTime := T#50ms);
        Dose : fillingcell::SK_Dose(UaRoot := "/Objects/Demo/Bench/Dose", UaEnable := FALSE, IoBackend := 0, Timeout := T#5s, UnitRunning := TRUE, P1 := 0.3);
        Caller : iec61499::events::E_CYCLE(DT := T#2s);
        Done : iec61499::events::E_CTU;
        Failed : iec61499::events::E_CTU;
      END_FBS
      EVENT_CONNECTIONS
        Boot.COLD TO Plant.INIT;
        Boot.WARM TO Plant.INIT;
        Boot.COLD TO PlantClock.START;
        Boot.WARM TO PlantClock.START;
        Boot.COLD TO Observer.INIT;
        Boot.WARM TO Observer.INIT;
        PlantClock.EO TO Plant.TICK;
        Plant.CNF TO Observer.SIM;
        Observer.INITO TO Dose.INIT;
        Dose.INITO TO Dose.UNIT_STAT;
        Dose.INITO TO Caller.START;
        Observer.SAMPLE TO Dose.SAMPLE;
        Caller.EO TO Dose.CALL;
        Dose.DONE TO Done.CU;
        Dose.DONE TO Plant.NEW_VIAL;
        Dose.FAILED TO Failed.CU;
      END_CONNECTIONS
      DATA_CONNECTIONS
        Plant.NeedleUp TO Observer.Sim_NeedleUp;
        Plant.NeedleDown TO Observer.Sim_NeedleDown;
        Plant.VialPresent TO Observer.Sim_VialPresent;
        Plant.FilledMl TO Observer.Sim_FilledMl;
        Plant.Stoppered TO Observer.Sim_Stoppered;
        Plant.Checked TO Observer.Sim_Checked;
        Plant.DoorClosed TO Observer.Sim_DoorClosed;
        Observer.Cell TO Dose.Cell;
        Dose.Drive TO Plant.DriveDose;
      END_CONNECTIONS
    END_RESOURCE
    RESOURCE PATTERNS : iec61499::system::EMB_RES
      FBS
        Boot : iec61499::events::E_RESTART;
        Clock : iec61499::events::E_CYCLE(DT := T#3s);
        Fork : fillingcell::P_Fork;
        WaitA : fillingcell::P_Wait(DT := T#300ms);
        WaitB : fillingcell::P_Wait(DT := T#800ms);
        Join : fillingcell::P_Join(N := 2);
        Loop : fillingcell::P_Loop(Count := 3);
        WaitC : fillingcell::P_Wait(DT := T#200ms);
        Toggle : iec61499::events::E_T_FF;
        Choice : fillingcell::P_Choice;
        CtuJoin : iec61499::events::E_CTU;
        CtuBody : iec61499::events::E_CTU;
        CtuTrue : iec61499::events::E_CTU;
        CtuFalse : iec61499::events::E_CTU;
      END_FBS
      EVENT_CONNECTIONS
        Boot.COLD TO Clock.START;
        Boot.WARM TO Clock.START;
        Clock.EO TO Fork.EI;
        Fork.EO1 TO WaitA.EI;
        Fork.EO2 TO WaitB.EI;
        WaitA.EO TO Join.EI1;
        WaitB.EO TO Join.EI2;
        Join.EO TO CtuJoin.CU;
        Join.EO TO Loop.EI;
        Loop.BODY TO WaitC.EI;
        Loop.BODY TO CtuBody.CU;
        WaitC.EO TO Loop.NEXT;
        Loop.EO TO Toggle.CLK;
        Toggle.EO TO Choice.EI;
        Choice.EO_TRUE TO CtuTrue.CU;
        Choice.EO_FALSE TO CtuFalse.CU;
      END_CONNECTIONS
      DATA_CONNECTIONS
        Toggle.Q TO Choice.Cond;
      END_CONNECTIONS
    END_RESOURCE
  END_DEVICE
  MAPPINGS
    FillingCell.Boot ON FORTE_PC.RES.Boot;
    FillingCell.Observer ON FORTE_PC.RES.Observer;
    FillingCell.UaFacade ON FORTE_PC.RES.UaFacade;
    FillingCell.Occupation ON FORTE_PC.RES.Occupation;
    FillingCell.Unit ON FORTE_PC.RES.Unit;
    FillingCell.Facade ON FORTE_PC.RES.Facade;
    FillingCell.EM_Filler ON FORTE_PC.RES.EM_Filler;
    FillingCell.PROC ON FORTE_PC.RES.PROC;
    FillingCellDemo.Boot ON FORTE_PC.DEMO.Boot;
    FillingCellDemo.Observer ON FORTE_PC.DEMO.Observer;
    FillingCellDemo.Occupation ON FORTE_PC.DEMO.Occupation;
    FillingCellDemo.Unit ON FORTE_PC.DEMO.Unit;
    FillingCellDemo.Facade ON FORTE_PC.DEMO.Facade;
    FillingCellDemo.EM_Filler ON FORTE_PC.DEMO.EM_Filler;
    FillingCellDemo.PROC ON FORTE_PC.DEMO.PROC;
    FillingCellDemo.Plant ON FORTE_PC.DEMO.Plant;
    FillingCellDemo.PlantClock ON FORTE_PC.DEMO.PlantClock;
    FillingCellDemo.Operator ON FORTE_PC.DEMO.Operator;
    FillingCellDemo.OpDelay ON FORTE_PC.DEMO.OpDelay;
    SkillBench.Boot ON FORTE_PC.BENCH.Boot;
    SkillBench.Plant ON FORTE_PC.BENCH.Plant;
    SkillBench.PlantClock ON FORTE_PC.BENCH.PlantClock;
    SkillBench.Observer ON FORTE_PC.BENCH.Observer;
    SkillBench.Dose ON FORTE_PC.BENCH.Dose;
    SkillBench.Caller ON FORTE_PC.BENCH.Caller;
    SkillBench.Done ON FORTE_PC.BENCH.Done;
    SkillBench.Failed ON FORTE_PC.BENCH.Failed;
    PatternDemo.Boot ON FORTE_PC.PATTERNS.Boot;
    PatternDemo.Clock ON FORTE_PC.PATTERNS.Clock;
    PatternDemo.Fork ON FORTE_PC.PATTERNS.Fork;
    PatternDemo.WaitA ON FORTE_PC.PATTERNS.WaitA;
    PatternDemo.WaitB ON FORTE_PC.PATTERNS.WaitB;
    PatternDemo.Join ON FORTE_PC.PATTERNS.Join;
    PatternDemo.Loop ON FORTE_PC.PATTERNS.Loop;
    PatternDemo.WaitC ON FORTE_PC.PATTERNS.WaitC;
    PatternDemo.Toggle ON FORTE_PC.PATTERNS.Toggle;
    PatternDemo.Choice ON FORTE_PC.PATTERNS.Choice;
    PatternDemo.CtuJoin ON FORTE_PC.PATTERNS.CtuJoin;
    PatternDemo.CtuBody ON FORTE_PC.PATTERNS.CtuBody;
    PatternDemo.CtuTrue ON FORTE_PC.PATTERNS.CtuTrue;
    PatternDemo.CtuFalse ON FORTE_PC.PATTERNS.CtuFalse;
  END_MAPPINGS
END_SYSTEM
